LIN {X 0,Y 523.97,Z 254.844,A -85,B 0,C 180,E1 -4887.998,E2 -4887.998} C_VEL
LIN {X 0,Y 523.943,Z 254.846,A -85,B 0,C 180,E1 -4890.854,E2 -4890.854} C_VEL
LIN {X 0,Y 523.959,Z 254.847,A -85,B 0,C 180,E1 -4893.734,E2 -4893.734} C_VEL
LIN {X 0,Y 523.92,Z 254.85,A -85,B 0,C 180,E1 -4896.403,E2 -4896.403} C_VEL
LIN {X 0,Y 523.92,Z 254.85,A -85,B 0,C 180,E1 -4899.083,E2 -4899.083} C_VEL
LIN {X 0,Y 523.953,Z 254.847,A -85,B 0,C 180,E1 -4902.117,E2 -4902.117} C_VEL
LIN {X 0,Y 523.951,Z 254.848,A -85,B 0,C 180,E1 -4905.307,E2 -4905.307} C_VEL
LIN {X 0,Y 523.918,Z 254.849,A -85,B 0,C 180,E1 -4906.91,E2 -4906.91} C_VEL
LIN {X 0,Y 523.255,Z 254.934,A -85,B 0,C 180,E1 -4907.551,E2 -4907.551} C_VEL
LIN {X 0,Y 520.425,Z 255.289,A -85,B 0,C 180,E1 -4908.593,E2 -4908.593} C_VEL
LIN {X 0,Y 518.027,Z 255.589,A -85,B 0,C 180,E1 -4909.432,E2 -4909.432} C_VEL
LIN {X 0,Y 516.986,Z 255.716,A -85,B 0,C 180,E1 -4910.08,E2 -4910.08} C_VEL
LIN {X 0,Y 516.896,Z 255.726,A -85,B 0,C 180,E1 -4910.299,E2 -4910.299} C_VEL
LIN {X 0,Y 516.879,Z 255.727,A -85,B 0,C 180,E1 -4913.34,E2 -4913.34} C_VEL
LIN {X 0,Y 516.905,Z 255.724,A -85,B 0,C 180,E1 -4916.12,E2 -4916.12} C_VEL
LIN {X 0,Y 516.887,Z 255.727,A -85,B 0,C 180,E1 -4918.934,E2 -4918.934} C_VEL
LIN {X 0,Y 516.917,Z 255.723,A -85,B 0,C 180,E1 -4921.584,E2 -4921.584} C_VEL
LIN {X 0,Y 516.925,Z 255.721,A -85,B 0,C 180,E1 -4924.21,E2 -4924.21} C_VEL
LIN {X 0,Y 516.863,Z 255.727,A -85,B 0,C 180,E1 -4926.776,E2 -4926.776} C_VEL
LIN {X 0,Y 516.93,Z 255.721,A -85,B 0,C 180,E1 -4929.73,E2 -4929.73} C_VEL
LIN {X 0,Y 516.922,Z 255.722,A -85,B 0,C 180,E1 -4932.595,E2 -4932.595} C_VEL
LIN {X 0,Y 516.94,Z 255.719,A -85,B 0,C 180,E1 -4935.03,E2 -4935.03} C_VEL
LIN {X 0,Y 516.994,Z 255.712,A -85,B 0,C 180,E1 -4938.234,E2 -4938.234} C_VEL
LIN {X 0,Y 516.964,Z 255.717,A -85,B 0,C 180,E1 -4941.399,E2 -4941.399} C_VEL
LIN {X 0,Y 517.001,Z 255.713,A -85,B 0,C 180,E1 -4943.756,E2 -4943.756} C_VEL
LIN {X 0,Y 516.718,Z 255.749,A -85,B 0,C 180,E1 -4946.1,E2 -4946.1} C_VEL
LIN {X 0,Y 516.592,Z 255.877,A -85,B 0,C 180,E1 -4947.66,E2 -4947.66} C_VEL
LIN {X 0,Y 516.81,Z 258.103,A -85,B 0,C 180,E1 -4949.999,E2 -4949.999} C_VEL
LIN {X 0,Y 516.55,Z 261.858,A -85,B 0,C 180,E1 -4953.9,E2 -4953.9} C_VEL
LIN {X 0,Y 516.473,Z 264.87,A -85,B 0,C 180,E1 -4957.034,E2 -4957.034} C_VEL
LIN {X 0,Y 516.409,Z 267.914,A -85,B 0,C 180,E1 -4960.19,E2 -4960.19} C_VEL
LIN {X 0,Y 516.387,Z 270.207,A -85,B 0,C 180,E1 -4962.577,E2 -4962.577} C_VEL
LIN {X 0,Y 516.346,Z 271.07,A -85,B 0,C 180,E1 -4963.453,E2 -4963.453} C_VEL
LIN {X 0,Y 520.193,Z 284.754,A -85,B 0,C 180,E1 -4963.9,E2 -4963.9} C_VEL
LIN {X 0,Y 520.737,Z 287.139,A -85,B 0,C 180,E1 -4963.984,E2 -4963.984} C_VEL
LIN {X 0,Y 520.379,Z 301.279,A -85,B 0,C 180,E1 -4964.418,E2 -4964.418} C_VEL
LIN {X 0,Y 519.918,Z 315.967,A -85,B 0,C 180,E1 -4965.032,E2 -4965.032} C_VEL
LIN {X 0,Y 519.498,Z 328.44,A -85,B 0,C 180,E1 -4965.697,E2 -4965.697} C_VEL
LIN {X 0,Y 519.047,Z 341.031,A -85,B 0,C 180,E1 -4966.519,E2 -4966.519} C_VEL
LIN {X 0,Y 518.554,Z 352.891,A -85,B 0,C 180,E1 -4967.449,E2 -4967.449} C_VEL
LIN {X 0,Y 518.04,Z 364.714,A -85,B 0,C 180,E1 -4968.557,E2 -4968.557} C_VEL
LIN {X 0,Y 517.549,Z 376.157,A -85,B 0,C 180,E1 -4969.845,E2 -4969.845} C_VEL
LIN {X 0,Y 517.19,Z 385.528,A -85,B 0,C 180,E1 -4971.106,E2 -4971.106} C_VEL
LIN {X 0,Y 516.848,Z 394.593,A -85,B 0,C 180,E1 -4972.568,E2 -4972.568} C_VEL
LIN {X 0,Y 516.611,Z 402.308,A -85,B 0,C 180,E1 -4974.086,E2 -4974.086} C_VEL
LIN {X 0,Y 516.475,Z 407.75,A -85,B 0,C 180,E1 -4975.381,E2 -4975.381} C_VEL
LIN {X 0,Y 516.327,Z 413.495,A -85,B 0,C 180,E1 -4977.128,E2 -4977.128} C_VEL
LIN {X 0,Y 516.24,Z 416.777,A -85,B 0,C 180,E1 -4978.455,E2 -4978.455} C_VEL
LIN {X 0,Y 516.227,Z 418.584,A -85,B 0,C 180,E1 -4979.392,E2 -4979.392} C_VEL
LIN {X 0,Y 516.165,Z 420.848,A -85,B 0,C 180,E1 -4981.157,E2 -4981.157} C_VEL
LIN {X 0,Y 516.166,Z 421.563,A -85,B 0,C 180,E1 -4982.419,E2 -4982.419} C_VEL
LIN {X 0,Y 516.163,Z 421.505,A -85,B 0,C 180,E1 -4983.934,E2 -4983.934} C_VEL
LIN {X 0,Y 516.161,Z 420.566,A -85,B 0,C 180,E1 -4985.221,E2 -4985.221} C_VEL
LIN {X 0,Y 516.178,Z 418.411,A -85,B 0,C 180,E1 -4986.803,E2 -4986.803} C_VEL
LIN {X 0,Y 516.31,Z 415.336,A -85,B 0,C 180,E1 -4988.277,E2 -4988.277} C_VEL
LIN {X 0,Y 516.374,Z 411.065,A -85,B 0,C 180,E1 -4989.767,E2 -4989.767} C_VEL
LIN {X 0,Y 516.469,Z 405.957,A -85,B 0,C 180,E1 -4991.167,E2 -4991.167} C_VEL
LIN {X 0,Y 516.694,Z 398.838,A -85,B 0,C 180,E1 -4992.737,E2 -4992.737} C_VEL
LIN {X 0,Y 517.005,Z 390.921,A -85,B 0,C 180,E1 -4994.159,E2 -4994.159} C_VEL
LIN {X 0,Y 517.345,Z 381.995,A -85,B 0,C 180,E1 -4995.497,E2 -4995.497} C_VEL
LIN {X 0,Y 517.719,Z 372.189,A -85,B 0,C 180,E1 -4996.735,E2 -4996.735} C_VEL
LIN {X 0,Y 518.239,Z 360.952,A -85,B 0,C 180,E1 -4997.922,E2 -4997.922} C_VEL
LIN {X 0,Y 518.715,Z 350.053,A -85,B 0,C 180,E1 -4998.895,E2 -4998.895} C_VEL
LIN {X 0,Y 519.286,Z 336.91,A -85,B 0,C 180,E1 -4999.87,E2 -4999.87} C_VEL
LIN {X 0,Y 519.784,Z 322.543,A -85,B 0,C 180,E1 -5000.734,E2 -5000.734} C_VEL
LIN {X 0,Y 520.24,Z 308.093,A -85,B 0,C 180,E1 -5001.415,E2 -5001.415} C_VEL
LIN {X 0,Y 520.598,Z 293.591,A -85,B 0,C 180,E1 -5001.933,E2 -5001.933} C_VEL
LIN {X 0,Y 520.56,Z 286.17,A -85,B 0,C 180,E1 -5002.145,E2 -5002.145} C_VEL
LIN {X 0,Y 517.771,Z 276.119,A -85,B 0,C 180,E1 -5002.476,E2 -5002.476} C_VEL
LIN {X 0,Y 516.369,Z 271.47,A -85,B 0,C 180,E1 -5002.633,E2 -5002.633} C_VEL
LIN {X 0,Y 516.417,Z 269.147,A -85,B 0,C 180,E1 -5005.141,E2 -5005.141} C_VEL
LIN {X 0,Y 516.47,Z 266.567,A -85,B 0,C 180,E1 -5007.948,E2 -5007.948} C_VEL
LIN {X 0,Y 516.557,Z 264.068,A -85,B 0,C 180,E1 -5010.674,E2 -5010.674} C_VEL
LIN {X 0,Y 516.56,Z 261.657,A -85,B 0,C 180,E1 -5013.323,E2 -5013.323} C_VEL
LIN {X 0,Y 516.681,Z 259.257,A -85,B 0,C 180,E1 -5015.918,E2 -5015.918} C_VEL
LIN {X 0,Y 516.642,Z 256.888,A -85,B 0,C 180,E1 -5018.453,E2 -5018.453} C_VEL
LIN {X 0,Y 516.705,Z 255.752,A -85,B 0,C 180,E1 -5019.8,E2 -5019.8} C_VEL
LIN {X 0,Y 516.891,Z 255.729,A -85,B 0,C 180,E1 -5022.596,E2 -5022.596} C_VEL
LIN {X 0,Y 516.935,Z 255.721,A -85,B 0,C 180,E1 -5025.031,E2 -5025.031} C_VEL
LIN {X 0,Y 516.959,Z 255.717,A -85,B 0,C 180,E1 -5028.235,E2 -5028.235} C_VEL
LIN {X 0,Y 516.965,Z 255.716,A -85,B 0,C 180,E1 -5031.401,E2 -5031.401} C_VEL
LIN {X 0,Y 517.006,Z 255.712,A -85,B 0,C 180,E1 -5033.758,E2 -5033.758} C_VEL
LIN {X 0,Y 517.081,Z 255.701,A -85,B 0,C 180,E1 -5037.664,E2 -5037.664} C_VEL
LIN {X 0,Y 517.09,Z 255.701,A -85,B 0,C 180,E1 -5040.78,E2 -5040.78} C_VEL
LIN {X 0,Y 517.011,Z 255.711,A -85,B 0,C 180,E1 -5043.118,E2 -5043.118} C_VEL
LIN {X 0,Y 517.007,Z 255.71,A -85,B 0,C 180,E1 -5046.244,E2 -5046.244} C_VEL
LIN {X 0,Y 516.953,Z 255.718,A -85,B 0,C 180,E1 -5049.39,E2 -5049.39} C_VEL
LIN {X 0,Y 516.949,Z 255.719,A -85,B 0,C 180,E1 -5051.808,E2 -5051.808} C_VEL
LIN {X 0,Y 516.941,Z 255.719,A -85,B 0,C 180,E1 -5055.147,E2 -5055.147} C_VEL
LIN {X 0,Y 516.922,Z 255.723,A -85,B 0,C 180,E1 -5058.223,E2 -5058.223} C_VEL
LIN {X 0,Y 516.911,Z 255.723,A -85,B 0,C 180,E1 -5060.702,E2 -5060.702} C_VEL
LIN {X 0,Y 516.909,Z 255.723,A -85,B 0,C 180,E1 -5064.073,E2 -5064.073} C_VEL
LIN {X 0,Y 516.927,Z 255.723,A -85,B 0,C 180,E1 -5066.658,E2 -5066.658} C_VEL
LIN {X 0,Y 516.909,Z 255.725,A -85,B 0,C 180,E1 -5069.524,E2 -5069.524} C_VEL
LIN {X 0,Y 516.893,Z 255.728,A -85,B 0,C 180,E1 -5072.544,E2 -5072.544} C_VEL
LIN {X 0,Y 516.864,Z 255.733,A -85,B 0,C 180,E1 -5075.33,E2 -5075.33} C_VEL
LIN {X 0,Y 516.879,Z 255.73,A -85,B 0,C 180,E1 -5077.944,E2 -5077.944} C_VEL
LIN {X 0,Y 516.883,Z 255.729,A -85,B 0,C 180,E1 -5080.742,E2 -5080.742} C_VEL
LIN {X 0,Y 516.882,Z 255.729,A -85,B 0,C 180,E1 -5082.832,E2 -5082.832} C_VEL
LIN {X 0,Y 516.93,Z 255.773,A -85,B 0,C 180,E1 -5084.578,E2 -5084.578} C_VEL
LIN {X 0,Y 517.92,Z 261.24,A -85,B 0,C 180,E1 -5087.119,E2 -5087.119} C_VEL
LIN {X 0,Y 518.273,Z 265.231,A -85,B 0,C 180,E1 -5088.878,E2 -5088.878} C_VEL
LIN {X 0,Y 518.125,Z 271.563,A -85,B 0,C 180,E1 -5091.395,E2 -5091.395} C_VEL
LIN {X 0,Y 517.889,Z 277.824,A -85,B 0,C 180,E1 -5093.821,E2 -5093.821} C_VEL
LIN {X 0,Y 517.701,Z 286.966,A -85,B 0,C 180,E1 -5097.112,E2 -5097.112} C_VEL
LIN {X 0,Y 517.53,Z 294.866,A -85,B 0,C 180,E1 -5099.838,E2 -5099.838} C_VEL
LIN {X 0,Y 517.327,Z 302.394,A -85,B 0,C 180,E1 -5102.491,E2 -5102.491} C_VEL
LIN {X 0,Y 517.143,Z 309.82,A -85,B 0,C 180,E1 -5105.085,E2 -5105.085} C_VEL
LIN {X 0,Y 516.963,Z 318.485,A -85,B 0,C 180,E1 -5108.047,E2 -5108.047} C_VEL
LIN {X 0,Y 516.826,Z 325.427,A -85,B 0,C 180,E1 -5110.378,E2 -5110.378} C_VEL
LIN {X 0,Y 520.774,Z 341.818,A -85,B 0,C 180,E1 -5110.836,E2 -5110.836} C_VEL
LIN {X 0,Y 520.392,Z 356.97,A -85,B 0,C 180,E1 -5111.264,E2 -5111.264} C_VEL
LIN {X 0,Y 520.029,Z 371.072,A -85,B 0,C 180,E1 -5111.817,E2 -5111.817} C_VEL
LIN {X 0,Y 519.548,Z 384.377,A -85,B 0,C 180,E1 -5112.484,E2 -5112.484} C_VEL
LIN {X 0,Y 519.048,Z 397.209,A -85,B 0,C 180,E1 -5113.279,E2 -5113.279} C_VEL
LIN {X 0,Y 518.531,Z 410.363,A -85,B 0,C 180,E1 -5114.272,E2 -5114.272} C_VEL
LIN {X 0,Y 518.039,Z 421.386,A -85,B 0,C 180,E1 -5115.264,E2 -5115.264} C_VEL
LIN {X 0,Y 517.634,Z 432.514,A -85,B 0,C 180,E1 -5116.456,E2 -5116.456} C_VEL
LIN {X 0,Y 517.156,Z 443.311,A -85,B 0,C 180,E1 -5117.841,E2 -5117.841} C_VEL
LIN {X 0,Y 516.912,Z 452.298,A -85,B 0,C 180,E1 -5119.226,E2 -5119.226} C_VEL
LIN {X 0,Y 516.637,Z 459.753,A -85,B 0,C 180,E1 -5120.606,E2 -5120.606} C_VEL
LIN {X 0,Y 516.463,Z 466.703,A -85,B 0,C 180,E1 -5122.18,E2 -5122.18} C_VEL
LIN {X 0,Y 516.36,Z 472.164,A -85,B 0,C 180,E1 -5123.75,E2 -5123.75} C_VEL
LIN {X 0,Y 516.239,Z 476.293,A -85,B 0,C 180,E1 -5125.315,E2 -5125.315} C_VEL
LIN {X 0,Y 516.272,Z 479.187,A -85,B 0,C 180,E1 -5126.879,E2 -5126.879} C_VEL
LIN {X 0,Y 516.189,Z 480.911,A -85,B 0,C 180,E1 -5128.44,E2 -5128.44} C_VEL
LIN {X 0,Y 516.151,Z 481.5,A -85,B 0,C 180,E1 -5130.001,E2 -5130.001} C_VEL
LIN {X 0,Y 516.189,Z 480.909,A -85,B 0,C 180,E1 -5131.561,E2 -5131.561} C_VEL
LIN {X 0,Y 516.272,Z 479.182,A -85,B 0,C 180,E1 -5133.122,E2 -5133.122} C_VEL
LIN {X 0,Y 516.239,Z 476.289,A -85,B 0,C 180,E1 -5134.686,E2 -5134.686} C_VEL
LIN {X 0,Y 516.352,Z 472.163,A -85,B 0,C 180,E1 -5136.252,E2 -5136.252} C_VEL
LIN {X 0,Y 516.464,Z 466.699,A -85,B 0,C 180,E1 -5137.822,E2 -5137.822} C_VEL
LIN {X 0,Y 516.638,Z 459.744,A -85,B 0,C 180,E1 -5139.396,E2 -5139.396} C_VEL
LIN {X 0,Y 516.973,Z 451.082,A -85,B 0,C 180,E1 -5140.972,E2 -5140.972} C_VEL
LIN {X 0,Y 517.228,Z 442.019,A -85,B 0,C 180,E1 -5142.338,E2 -5142.338} C_VEL
LIN {X 0,Y 517.635,Z 432.504,A -85,B 0,C 180,E1 -5143.545,E2 -5143.545} C_VEL
LIN {X 0,Y 518.095,Z 420.35,A -85,B 0,C 180,E1 -5144.836,E2 -5144.836} C_VEL
LIN {X 0,Y 518.628,Z 408.21,A -85,B 0,C 180,E1 -5145.907,E2 -5145.907} C_VEL
LIN {X 0,Y 519.087,Z 395.767,A -85,B 0,C 180,E1 -5146.822,E2 -5146.822} C_VEL
LIN {X 0,Y 519.577,Z 382.586,A -85,B 0,C 180,E1 -5147.618,E2 -5147.618} C_VEL
LIN {X 0,Y 520.083,Z 369.43,A -85,B 0,C 180,E1 -5148.255,E2 -5148.255} C_VEL
LIN {X 0,Y 520.483,Z 354.499,A -85,B 0,C 180,E1 -5148.816,E2 -5148.816} C_VEL
LIN {X 0,Y 520.673,Z 341.239,A -85,B 0,C 180,E1 -5149.182,E2 -5149.182} C_VEL
LIN {X 0,Y 516.823,Z 325.426,A -85,B 0,C 180,E1 -5149.622,E2 -5149.622} C_VEL
LIN {X 0,Y 516.971,Z 317.119,A -85,B 0,C 180,E1 -5152.417,E2 -5152.417} C_VEL
LIN {X 0,Y 517.188,Z 308.579,A -85,B 0,C 180,E1 -5155.344,E2 -5155.344} C_VEL
LIN {X 0,Y 517.427,Z 299.915,A -85,B 0,C 180,E1 -5158.385,E2 -5158.385} C_VEL
LIN {X 0,Y 517.554,Z 291.891,A -85,B 0,C 180,E1 -5161.185,E2 -5161.185} C_VEL
LIN {X 0,Y 517.817,Z 283.8,A -85,B 0,C 180,E1 -5164.115,E2 -5164.115} C_VEL
LIN {X 0,Y 518.095,Z 275.662,A -85,B 0,C 180,E1 -5167.183,E2 -5167.183} C_VEL
LIN {X 0,Y 518.293,Z 268.202,A -85,B 0,C 180,E1 -5170.092,E2 -5170.092} C_VEL
LIN {X 0,Y 518.181,Z 263.095,A -85,B 0,C 180,E1 -5172.194,E2 -5172.194} C_VEL
LIN {X 0,Y 517.331,Z 257.986,A -85,B 0,C 180,E1 -5174.503,E2 -5174.503} C_VEL
LIN {X 0,Y 516.923,Z 255.721,A -85,B 0,C 180,E1 -5175.626,E2 -5175.626} C_VEL
LIN {X 0,Y 516.918,Z 255.724,A -85,B 0,C 180,E1 -5178.399,E2 -5178.399} C_VEL
LIN {X 0,Y 516.885,Z 255.727,A -85,B 0,C 180,E1 -5181.284,E2 -5181.284} C_VEL
LIN {X 0,Y 516.876,Z 255.727,A -85,B 0,C 180,E1 -5184.22,E2 -5184.22} C_VEL
LIN {X 0,Y 516.886,Z 255.727,A -85,B 0,C 180,E1 -5187.052,E2 -5187.052} C_VEL
LIN {X 0,Y 516.897,Z 255.725,A -85,B 0,C 180,E1 -5189.796,E2 -5189.796} C_VEL
LIN {X 0,Y 516.932,Z 255.721,A -85,B 0,C 180,E1 -5192.467,E2 -5192.467} C_VEL
LIN {X 0,Y 516.914,Z 255.724,A -85,B 0,C 180,E1 -5195.072,E2 -5195.072} C_VEL
LIN {X 0,Y 516.892,Z 255.727,A -85,B 0,C 180,E1 -5198.462,E2 -5198.462} C_VEL
LIN {X 0,Y 516.909,Z 255.724,A -85,B 0,C 180,E1 -5200.954,E2 -5200.954} C_VEL
LIN {X 0,Y 516.919,Z 255.722,A -85,B 0,C 180,E1 -5203.41,E2 -5203.41} C_VEL
LIN {X 0,Y 516.899,Z 255.725,A -85,B 0,C 180,E1 -5205.833,E2 -5205.833} C_VEL
LIN {X 0,Y 516.971,Z 255.716,A -85,B 0,C 180,E1 -5208.233,E2 -5208.233} C_VEL
LIN {X 0,Y 516.971,Z 255.715,A -85,B 0,C 180,E1 -5211.399,E2 -5211.399} C_VEL
LIN {X 0,Y 517.028,Z 255.709,A -85,B 0,C 180,E1 -5214.539,E2 -5214.539} C_VEL
LIN {X 0,Y 517.088,Z 255.7,A -85,B 0,C 180,E1 -5217.662,E2 -5217.662} C_VEL
LIN {X 0,Y 517.098,Z 255.7,A -85,B 0,C 180,E1 -5220.778,E2 -5220.778} C_VEL
LIN {X 0,Y 517.015,Z 255.711,A -85,B 0,C 180,E1 -5223.116,E2 -5223.116} C_VEL
LIN {X 0,Y 517.012,Z 255.711,A -85,B 0,C 180,E1 -5226.242,E2 -5226.242} C_VEL
LIN {X 0,Y 516.954,Z 255.717,A -85,B 0,C 180,E1 -5229.388,E2 -5229.388} C_VEL
LIN {X 0,Y 516.955,Z 255.719,A -85,B 0,C 180,E1 -5231.806,E2 -5231.806} C_VEL
LIN {X 0,Y 516.947,Z 255.717,A -85,B 0,C 180,E1 -5235.145,E2 -5235.145} C_VEL
LIN {X 0,Y 516.927,Z 255.722,A -85,B 0,C 180,E1 -5238.221,E2 -5238.221} C_VEL
LIN {X 0,Y 516.913,Z 255.723,A -85,B 0,C 180,E1 -5240.7,E2 -5240.7} C_VEL
LIN {X 0,Y 516.912,Z 255.724,A -85,B 0,C 180,E1 -5244.071,E2 -5244.071} C_VEL
LIN {X 0,Y 516.926,Z 255.721,A -85,B 0,C 180,E1 -5246.656,E2 -5246.656} C_VEL
LIN {X 0,Y 516.91,Z 255.724,A -85,B 0,C 180,E1 -5249.523,E2 -5249.523} C_VEL
LIN {X 0,Y 516.896,Z 255.726,A -85,B 0,C 180,E1 -5252.543,E2 -5252.543} C_VEL
LIN {X 0,Y 516.881,Z 255.726,A -85,B 0,C 180,E1 -5255.331,E2 -5255.331} C_VEL
LIN {X 0,Y 516.879,Z 255.729,A -85,B 0,C 180,E1 -5257.942,E2 -5257.942} C_VEL
LIN {X 0,Y 516.882,Z 255.727,A -85,B 0,C 180,E1 -5260.74,E2 -5260.74} C_VEL
LIN {X 0,Y 516.9,Z 255.724,A -85,B 0,C 180,E1 -5262.828,E2 -5262.828} C_VEL
LIN {X 0,Y 516.918,Z 255.722,A -85,B 0,C 180,E1 -5265.009,E2 -5265.009} C_VEL
LIN {X 0,Y 516.917,Z 255.722,A -85,B 0,C 180,E1 -5268.396,E2 -5268.396} C_VEL
LIN {X 0,Y 516.896,Z 255.726,A -85,B 0,C 180,E1 -5270.299,E2 -5270.299} C_VEL
LIN {X 0,Y 516.215,Z 255.809,A -85,B 0,C 180,E1 -5270.949,E2 -5270.949} C_VEL
LIN {X 0,Y 513.362,Z 256.166,A -85,B 0,C 180,E1 -5272.004,E2 -5272.004} C_VEL
LIN {X 0,Y 510.954,Z 256.469,A -85,B 0,C 180,E1 -5272.855,E2 -5272.855} C_VEL
LIN {X 0,Y 509.914,Z 256.597,A -85,B 0,C 180,E1 -5273.511,E2 -5273.511} C_VEL
LIN {X 0,Y 509.826,Z 256.607,A -85,B 0,C 180,E1 -5273.733,E2 -5273.733} C_VEL
LIN {X 0,Y 509.855,Z 256.602,A -85,B 0,C 180,E1 -5276.538,E2 -5276.538} C_VEL
LIN {X 0,Y 509.843,Z 256.604,A -85,B 0,C 180,E1 -5279.334,E2 -5279.334} C_VEL
LIN {X 0,Y 509.888,Z 256.598,A -85,B 0,C 180,E1 -5282.054,E2 -5282.054} C_VEL
LIN {X 0,Y 509.87,Z 256.599,A -85,B 0,C 180,E1 -5284.703,E2 -5284.703} C_VEL
LIN {X 0,Y 509.847,Z 256.604,A -85,B 0,C 180,E1 -5287.449,E2 -5287.449} C_VEL
LIN {X 0,Y 509.908,Z 256.596,A -85,B 0,C 180,E1 -5289.844,E2 -5289.844} C_VEL
LIN {X 0,Y 509.878,Z 256.6,A -85,B 0,C 180,E1 -5293.174,E2 -5293.174} C_VEL
LIN {X 0,Y 509.864,Z 256.602,A -85,B 0,C 180,E1 -5295.634,E2 -5295.634} C_VEL
LIN {X 0,Y 509.916,Z 256.595,A -85,B 0,C 180,E1 -5298.874,E2 -5298.874} C_VEL
LIN {X 0,Y 509.942,Z 256.59,A -85,B 0,C 180,E1 -5302.078,E2 -5302.078} C_VEL
LIN {X 0,Y 509.943,Z 256.589,A -85,B 0,C 180,E1 -5304.463,E2 -5304.463} C_VEL
LIN {X 0,Y 509.534,Z 256.645,A -85,B 0,C 180,E1 -5307.628,E2 -5307.628} C_VEL
LIN {X 0,Y 509.795,Z 258.058,A -85,B 0,C 180,E1 -5309.21,E2 -5309.21} C_VEL
LIN {X 0,Y 509.474,Z 260.352,A -85,B 0,C 180,E1 -5311.58,E2 -5311.58} C_VEL
LIN {X 0,Y 509.465,Z 263.372,A -85,B 0,C 180,E1 -5314.747,E2 -5314.747} C_VEL
LIN {X 0,Y 509.418,Z 265.644,A -85,B 0,C 180,E1 -5317.132,E2 -5317.132} C_VEL
LIN {X 0,Y 509.344,Z 268.73,A -85,B 0,C 180,E1 -5320.333,E2 -5320.333} C_VEL
LIN {X 0,Y 509.292,Z 271.48,A -85,B 0,C 180,E1 -5323.186,E2 -5323.186} C_VEL
LIN {X 0,Y 513.52,Z 286.197,A -85,B 0,C 180,E1 -5323.67,E2 -5323.67} C_VEL
LIN {X 0,Y 513.979,Z 288.927,A -85,B 0,C 180,E1 -5323.766,E2 -5323.766} C_VEL
LIN {X 0,Y 513.576,Z 304.035,A -85,B 0,C 180,E1 -5324.259,E2 -5324.259} C_VEL
LIN {X 0,Y 513.1,Z 318.162,A -85,B 0,C 180,E1 -5324.881,E2 -5324.881} C_VEL
LIN {X 0,Y 512.637,Z 331.194,A -85,B 0,C 180,E1 -5325.607,E2 -5325.607} C_VEL
LIN {X 0,Y 512.081,Z 345.219,A -85,B 0,C 180,E1 -5326.578,E2 -5326.578} C_VEL
LIN {X 0,Y 511.549,Z 357.293,A -85,B 0,C 180,E1 -5327.592,E2 -5327.592} C_VEL
LIN {X 0,Y 511.012,Z 367.896,A -85,B 0,C 180,E1 -5328.648,E2 -5328.648} C_VEL
LIN {X 0,Y 510.55,Z 378.603,A -85,B 0,C 180,E1 -5329.919,E2 -5329.919} C_VEL
LIN {X 0,Y 510.119,Z 387.673,A -85,B 0,C 180,E1 -5331.201,E2 -5331.201} C_VEL
LIN {X 0,Y 509.798,Z 396.556,A -85,B 0,C 180,E1 -5332.705,E2 -5332.705} C_VEL
LIN {X 0,Y 509.575,Z 402.926,A -85,B 0,C 180,E1 -5334.007,E2 -5334.007} C_VEL
LIN {X 0,Y 509.418,Z 408.335,A -85,B 0,C 180,E1 -5335.32,E2 -5335.32} C_VEL
LIN {X 0,Y 509.287,Z 412.746,A -85,B 0,C 180,E1 -5336.646,E2 -5336.646} C_VEL
LIN {X 0,Y 509.195,Z 416.312,A -85,B 0,C 180,E1 -5337.986,E2 -5337.986} C_VEL
LIN {X 0,Y 509.131,Z 419.721,A -85,B 0,C 180,E1 -5339.797,E2 -5339.797} C_VEL
LIN {X 0,Y 509.089,Z 421.296,A -85,B 0,C 180,E1 -5341.142,E2 -5341.142} C_VEL
LIN {X 0,Y 509.072,Z 422.049,A -85,B 0,C 180,E1 -5342.636,E2 -5342.636} C_VEL
LIN {X 0,Y 509.095,Z 421.64,A -85,B 0,C 180,E1 -5344.471,E2 -5344.471} C_VEL
LIN {X 0,Y 509.073,Z 420.803,A -85,B 0,C 180,E1 -5345.462,E2 -5345.462} C_VEL
LIN {X 0,Y 509.109,Z 418.94,A -85,B 0,C 180,E1 -5346.809,E2 -5346.809} C_VEL
LIN {X 0,Y 509.251,Z 415.678,A -85,B 0,C 180,E1 -5348.39,E2 -5348.39} C_VEL
LIN {X 0,Y 509.34,Z 411.357,A -85,B 0,C 180,E1 -5349.912,E2 -5349.912} C_VEL
LIN {X 0,Y 509.461,Z 405.675,A -85,B 0,C 180,E1 -5351.464,E2 -5351.464} C_VEL
LIN {X 0,Y 509.715,Z 398.396,A -85,B 0,C 180,E1 -5353.051,E2 -5353.051} C_VEL
LIN {X 0,Y 510.048,Z 390.848,A -85,B 0,C 180,E1 -5354.399,E2 -5354.399} C_VEL
LIN {X 0,Y 510.428,Z 382.045,A -85,B 0,C 180,E1 -5355.723,E2 -5355.723} C_VEL
LIN {X 0,Y 510.86,Z 371.824,A -85,B 0,C 180,E1 -5357.014,E2 -5357.014} C_VEL
LIN {X 0,Y 511.407,Z 360.57,A -85,B 0,C 180,E1 -5358.204,E2 -5358.204} C_VEL
LIN {X 0,Y 511.945,Z 349.159,A -85,B 0,C 180,E1 -5359.218,E2 -5359.218} C_VEL
LIN {X 0,Y 512.5,Z 336.309,A -85,B 0,C 180,E1 -5360.168,E2 -5360.168} C_VEL
LIN {X 0,Y 513.037,Z 323.002,A -85,B 0,C 180,E1 -5360.971,E2 -5360.971} C_VEL
LIN {X 0,Y 513.52,Z 308.765,A -85,B 0,C 180,E1 -5361.652,E2 -5361.652} C_VEL
LIN {X 0,Y 513.923,Z 293.692,A -85,B 0,C 180,E1 -5362.196,E2 -5362.196} C_VEL
LIN {X 0,Y 513.81,Z 287.32,A -85,B 0,C 180,E1 -5362.384,E2 -5362.384} C_VEL
LIN {X 0,Y 510.983,Z 277.314,A -85,B 0,C 180,E1 -5362.73,E2 -5362.73} C_VEL
LIN {X 0,Y 509.309,Z 271.968,A -85,B 0,C 180,E1 -5362.903,E2 -5362.903} C_VEL
LIN {X 0,Y 509.363,Z 269.219,A -85,B 0,C 180,E1 -5365.878,E2 -5365.878} C_VEL
LIN {X 0,Y 509.457,Z 266.557,A -85,B 0,C 180,E1 -5368.791,E2 -5368.791} C_VEL
LIN {X 0,Y 509.499,Z 263.615,A -85,B 0,C 180,E1 -5372.032,E2 -5372.032} C_VEL
LIN {X 0,Y 509.542,Z 261.186,A -85,B 0,C 180,E1 -5374.687,E2 -5374.687} C_VEL
LIN {X 0,Y 509.59,Z 258.574,A -85,B 0,C 180,E1 -5377.521,E2 -5377.521} C_VEL
LIN {X 0,Y 509.677,Z 256.627,A -85,B 0,C 180,E1 -5379.836,E2 -5379.836} C_VEL
LIN {X 0,Y 509.855,Z 256.606,A -85,B 0,C 180,E1 -5382.348,E2 -5382.348} C_VEL
LIN {X 0,Y 509.903,Z 256.597,A -85,B 0,C 180,E1 -5384.82,E2 -5384.82} C_VEL
LIN {X 0,Y 509.895,Z 256.597,A -85,B 0,C 180,E1 -5388.124,E2 -5388.124} C_VEL
LIN {X 0,Y 509.912,Z 256.595,A -85,B 0,C 180,E1 -5391.281,E2 -5391.281} C_VEL
LIN {X 0,Y 509.974,Z 256.588,A -85,B 0,C 180,E1 -5393.671,E2 -5393.671} C_VEL
LIN {X 0,Y 510.052,Z 256.577,A -85,B 0,C 180,E1 -5397.632,E2 -5397.632} C_VEL
LIN {X 0,Y 510.06,Z 256.577,A -85,B 0,C 180,E1 -5400.79,E2 -5400.79} C_VEL
LIN {X 0,Y 509.953,Z 256.59,A -85,B 0,C 180,E1 -5403.161,E2 -5403.161} C_VEL
LIN {X 0,Y 509.975,Z 256.586,A -85,B 0,C 180,E1 -5406.33,E2 -5406.33} C_VEL
LIN {X 0,Y 509.914,Z 256.595,A -85,B 0,C 180,E1 -5408.721,E2 -5408.721} C_VEL
LIN {X 0,Y 509.901,Z 256.598,A -85,B 0,C 180,E1 -5411.932,E2 -5411.932} C_VEL
LIN {X 0,Y 509.891,Z 256.598,A -85,B 0,C 180,E1 -5415.243,E2 -5415.243} C_VEL
LIN {X 0,Y 509.885,Z 256.598,A -85,B 0,C 180,E1 -5418.002,E2 -5418.002} C_VEL
LIN {X 0,Y 509.849,Z 256.602,A -85,B 0,C 180,E1 -5421.002,E2 -5421.002} C_VEL
LIN {X 0,Y 509.835,Z 256.605,A -85,B 0,C 180,E1 -5423.564,E2 -5423.564} C_VEL
LIN {X 0,Y 509.912,Z 256.596,A -85,B 0,C 180,E1 -5426.38,E2 -5426.38} C_VEL
LIN {X 0,Y 509.875,Z 256.602,A -85,B 0,C 180,E1 -5428.845,E2 -5428.845} C_VEL
LIN {X 0,Y 509.817,Z 256.61,A -85,B 0,C 180,E1 -5431.591,E2 -5431.591} C_VEL
LIN {X 0,Y 509.845,Z 256.608,A -85,B 0,C 180,E1 -5434.414,E2 -5434.414} C_VEL
LIN {X 0,Y 509.815,Z 256.613,A -85,B 0,C 180,E1 -5437.341,E2 -5437.341} C_VEL
LIN {X 0,Y 509.836,Z 256.606,A -85,B 0,C 180,E1 -5440.383,E2 -5440.383} C_VEL
LIN {X 0,Y 509.822,Z 256.609,A -85,B 0,C 180,E1 -5443.063,E2 -5443.063} C_VEL
LIN {X 0,Y 509.859,Z 256.621,A -85,B 0,C 180,E1 -5444.212,E2 -5444.212} C_VEL
LIN {X 0,Y 510.86,Z 261.949,A -85,B 0,C 180,E1 -5446.814,E2 -5446.814} C_VEL
LIN {X 0,Y 511.314,Z 266.361,A -85,B 0,C 180,E1 -5448.719,E2 -5448.719} C_VEL
LIN {X 0,Y 511.148,Z 272.465,A -85,B 0,C 180,E1 -5451.23,E2 -5451.23} C_VEL
LIN {X 0,Y 510.909,Z 278.821,A -85,B 0,C 180,E1 -5453.737,E2 -5453.737} C_VEL
LIN {X 0,Y 510.676,Z 287.976,A -85,B 0,C 180,E1 -5457.087,E2 -5457.087} C_VEL
LIN {X 0,Y 510.47,Z 297.127,A -85,B 0,C 180,E1 -5460.289,E2 -5460.289} C_VEL
LIN {X 0,Y 510.293,Z 304.869,A -85,B 0,C 180,E1 -5462.968,E2 -5462.968} C_VEL
LIN {X 0,Y 510.057,Z 313.534,A -85,B 0,C 180,E1 -5466.017,E2 -5466.017} C_VEL
LIN {X 0,Y 509.883,Z 322.199,A -85,B 0,C 180,E1 -5469,E2 -5469} C_VEL
LIN {X 0,Y 509.781,Z 325.429,A -85,B 0,C 180,E1 -5470.096,E2 -5470.096} C_VEL
LIN {X 0,Y 513.785,Z 341.937,A -85,B 0,C 180,E1 -5470.567,E2 -5470.567} C_VEL
LIN {X 0,Y 513.991,Z 345.193,A -85,B 0,C 180,E1 -5470.657,E2 -5470.657} C_VEL
LIN {X 0,Y 513.657,Z 359.079,A -85,B 0,C 180,E1 -5471.081,E2 -5471.081} C_VEL
LIN {X 0,Y 513.169,Z 373.813,A -85,B 0,C 180,E1 -5471.692,E2 -5471.692} C_VEL
LIN {X 0,Y 512.613,Z 387.891,A -85,B 0,C 180,E1 -5472.446,E2 -5472.446} C_VEL
LIN {X 0,Y 512.032,Z 401.468,A -85,B 0,C 180,E1 -5473.351,E2 -5473.351} C_VEL
LIN {X 0,Y 511.536,Z 414.073,A -85,B 0,C 180,E1 -5474.376,E2 -5474.376} C_VEL
LIN {X 0,Y 510.962,Z 425.286,A -85,B 0,C 180,E1 -5475.463,E2 -5475.463} C_VEL
LIN {X 0,Y 510.504,Z 435.77,A -85,B 0,C 180,E1 -5476.669,E2 -5476.669} C_VEL
LIN {X 0,Y 510.002,Z 446.021,A -85,B 0,C 180,E1 -5478.071,E2 -5478.071} C_VEL
LIN {X 0,Y 509.818,Z 454.537,A -85,B 0,C 180,E1 -5479.476,E2 -5479.476} C_VEL
LIN {X 0,Y 509.536,Z 461.619,A -85,B 0,C 180,E1 -5480.874,E2 -5480.874} C_VEL
LIN {X 0,Y 509.352,Z 468.186,A -85,B 0,C 180,E1 -5482.469,E2 -5482.469} C_VEL
LIN {X 0,Y 509.297,Z 473.323,A -85,B 0,C 180,E1 -5484.06,E2 -5484.06} C_VEL
LIN {X 0,Y 509.159,Z 476.293,A -85,B 0,C 180,E1 -5485.25,E2 -5485.25} C_VEL
LIN {X 0,Y 509.188,Z 479.187,A -85,B 0,C 180,E1 -5486.836,E2 -5486.836} C_VEL
LIN {X 0,Y 509.11,Z 480.911,A -85,B 0,C 180,E1 -5488.418,E2 -5488.418} C_VEL
LIN {X 0,Y 509.063,Z 481.5,A -85,B 0,C 180,E1 -5490.001,E2 -5490.001} C_VEL
LIN {X 0,Y 509.11,Z 480.908,A -85,B 0,C 180,E1 -5491.583,E2 -5491.583} C_VEL
LIN {X 0,Y 509.189,Z 479.182,A -85,B 0,C 180,E1 -5493.165,E2 -5493.165} C_VEL
LIN {X 0,Y 509.159,Z 476.288,A -85,B 0,C 180,E1 -5494.751,E2 -5494.751} C_VEL
LIN {X 0,Y 509.262,Z 472.163,A -85,B 0,C 180,E1 -5496.339,E2 -5496.339} C_VEL
LIN {X 0,Y 509.386,Z 466.699,A -85,B 0,C 180,E1 -5497.931,E2 -5497.931} C_VEL
LIN {X 0,Y 509.561,Z 459.743,A -85,B 0,C 180,E1 -5499.527,E2 -5499.527} C_VEL
LIN {X 0,Y 509.956,Z 451.081,A -85,B 0,C 180,E1 -5501.125,E2 -5501.125} C_VEL
LIN {X 0,Y 510.24,Z 442.019,A -85,B 0,C 180,E1 -5502.51,E2 -5502.51} C_VEL
LIN {X 0,Y 510.654,Z 432.504,A -85,B 0,C 180,E1 -5503.734,E2 -5503.734} C_VEL
LIN {X 0,Y 511.181,Z 420.35,A -85,B 0,C 180,E1 -5505.041,E2 -5505.041} C_VEL
LIN {X 0,Y 511.747,Z 408.211,A -85,B 0,C 180,E1 -5506.127,E2 -5506.127} C_VEL
LIN {X 0,Y 512.274,Z 395.766,A -85,B 0,C 180,E1 -5507.053,E2 -5507.053} C_VEL
LIN {X 0,Y 512.789,Z 382.585,A -85,B 0,C 180,E1 -5507.859,E2 -5507.859} C_VEL
LIN {X 0,Y 513.399,Z 367.969,A -85,B 0,C 180,E1 -5508.568,E2 -5508.568} C_VEL
LIN {X 0,Y 513.798,Z 352.709,A -85,B 0,C 180,E1 -5509.131,E2 -5509.131} C_VEL
LIN {X 0,Y 513.944,Z 342.545,A -85,B 0,C 180,E1 -5509.413,E2 -5509.413} C_VEL
LIN {X 0,Y 509.999,Z 326.691,A -85,B 0,C 180,E1 -5509.876,E2 -5509.876} C_VEL
LIN {X 0,Y 509.8,Z 325.391,A -85,B 0,C 180,E1 -5509.916,E2 -5509.916} C_VEL
LIN {X 0,Y 509.929,Z 317.244,A -85,B 0,C 180,E1 -5512.7,E2 -5512.7} C_VEL
LIN {X 0,Y 510.188,Z 308.579,A -85,B 0,C 180,E1 -5515.717,E2 -5515.717} C_VEL
LIN {X 0,Y 510.46,Z 299.825,A -85,B 0,C 180,E1 -5518.809,E2 -5518.809} C_VEL
LIN {X 0,Y 510.634,Z 290.651,A -85,B 0,C 180,E1 -5521.998,E2 -5521.998} C_VEL
LIN {X 0,Y 510.854,Z 283.125,A -85,B 0,C 180,E1 -5524.815,E2 -5524.815} C_VEL
LIN {X 0,Y 511.174,Z 275.557,A -85,B 0,C 180,E1 -5527.722,E2 -5527.722} C_VEL
LIN {X 0,Y 511.322,Z 269.211,A -85,B 0,C 180,E1 -5530.241,E2 -5530.241} C_VEL
LIN {X 0,Y 511.208,Z 264.256,A -85,B 0,C 180,E1 -5532.349,E2 -5532.349} C_VEL
LIN {X 0,Y 510.351,Z 259.311,A -85,B 0,C 180,E1 -5534.614,E2 -5534.614} C_VEL
LIN {X 0,Y 509.86,Z 256.599,A -85,B 0,C 180,E1 -5535.941,E2 -5535.941} C_VEL
LIN {X 0,Y 509.86,Z 256.603,A -85,B 0,C 180,E1 -5538.574,E2 -5538.574} C_VEL
LIN {X 0,Y 509.856,Z 256.603,A -85,B 0,C 180,E1 -5541.786,E2 -5541.786} C_VEL
LIN {X 0,Y 509.835,Z 256.607,A -85,B 0,C 180,E1 -5544.622,E2 -5544.622} C_VEL
LIN {X 0,Y 509.865,Z 256.601,A -85,B 0,C 180,E1 -5547.481,E2 -5547.481} C_VEL
LIN {X 0,Y 509.864,Z 256.601,A -85,B 0,C 180,E1 -5550.274,E2 -5550.274} C_VEL
LIN {X 0,Y 509.89,Z 256.6,A -85,B 0,C 180,E1 -5552.944,E2 -5552.944} C_VEL
LIN {X 0,Y 509.87,Z 256.599,A -85,B 0,C 180,E1 -5555.573,E2 -5555.573} C_VEL
LIN {X 0,Y 509.856,Z 256.603,A -85,B 0,C 180,E1 -5558.998,E2 -5558.998} C_VEL
LIN {X 0,Y 509.895,Z 256.596,A -85,B 0,C 180,E1 -5561.999,E2 -5561.999} C_VEL
LIN {X 0,Y 509.916,Z 256.595,A -85,B 0,C 180,E1 -5564.818,E2 -5564.818} C_VEL
LIN {X 0,Y 509.906,Z 256.596,A -85,B 0,C 180,E1 -5568.124,E2 -5568.124} C_VEL
LIN {X 0,Y 509.917,Z 256.593,A -85,B 0,C 180,E1 -5571.279,E2 -5571.279} C_VEL
LIN {X 0,Y 509.978,Z 256.587,A -85,B 0,C 180,E1 -5574.463,E2 -5574.463} C_VEL
LIN {X 0,Y 510.059,Z 256.575,A -85,B 0,C 180,E1 -5577.63,E2 -5577.63} C_VEL
LIN {X 0,Y 510.069,Z 256.576,A -85,B 0,C 180,E1 -5580.789,E2 -5580.789} C_VEL
LIN {X 0,Y 509.957,Z 256.589,A -85,B 0,C 180,E1 -5583.159,E2 -5583.159} C_VEL
LIN {X 0,Y 509.981,Z 256.588,A -85,B 0,C 180,E1 -5586.329,E2 -5586.329} C_VEL
LIN {X 0,Y 509.917,Z 256.594,A -85,B 0,C 180,E1 -5588.719,E2 -5588.719} C_VEL
LIN {X 0,Y 509.907,Z 256.597,A -85,B 0,C 180,E1 -5591.931,E2 -5591.931} C_VEL
LIN {X 0,Y 509.896,Z 256.595,A -85,B 0,C 180,E1 -5595.241,E2 -5595.241} C_VEL
LIN {X 0,Y 509.89,Z 256.6,A -85,B 0,C 180,E1 -5598,E2 -5598} C_VEL
LIN {X 0,Y 509.851,Z 256.602,A -85,B 0,C 180,E1 -5601,E2 -5601} C_VEL
LIN {X 0,Y 509.87,Z 256.601,A -85,B 0,C 180,E1 -5604.425,E2 -5604.425} C_VEL
LIN {X 0,Y 509.885,Z 256.597,A -85,B 0,C 180,E1 -5607.054,E2 -5607.054} C_VEL
LIN {X 0,Y 509.856,Z 256.603,A -85,B 0,C 180,E1 -5609.75,E2 -5609.75} C_VEL
LIN {X 0,Y 509.873,Z 256.599,A -85,B 0,C 180,E1 -5612.773,E2 -5612.773} C_VEL
LIN {X 0,Y 509.84,Z 256.604,A -85,B 0,C 180,E1 -5615.58,E2 -5615.58} C_VEL
LIN {X 0,Y 509.848,Z 256.603,A -85,B 0,C 180,E1 -5618.337,E2 -5618.337} C_VEL
LIN {X 0,Y 509.855,Z 256.602,A -85,B 0,C 180,E1 -5621.424,E2 -5621.424} C_VEL
LIN {X 0,Y 509.852,Z 256.601,A -85,B 0,C 180,E1 -5624.667,E2 -5624.667} C_VEL
LIN {X 0,Y 509.876,Z 256.601,A -85,B 0,C 180,E1 -5628.099,E2 -5628.099} C_VEL
LIN {X 0,Y 509.854,Z 256.601,A -85,B 0,C 180,E1 -5630.648,E2 -5630.648} C_VEL
LIN {X 0,Y 509.826,Z 256.607,A -85,B 0,C 180,E1 -5633.733,E2 -5633.733} C_VEL
LIN {X 0,Y 509.159,Z 256.689,A -85,B 0,C 180,E1 -5634.393,E2 -5634.393} C_VEL
LIN {X 0,Y 506.341,Z 257.041,A -85,B 0,C 180,E1 -5635.465,E2 -5635.465} C_VEL
LIN {X 0,Y 503.948,Z 257.339,A -85,B 0,C 180,E1 -5636.328,E2 -5636.328} C_VEL
LIN {X 0,Y 502.9,Z 257.469,A -85,B 0,C 180,E1 -5636.995,E2 -5636.995} C_VEL
LIN {X 0,Y 502.802,Z 257.479,A -85,B 0,C 180,E1 -5637.22,E2 -5637.22} C_VEL
LIN {X 0,Y 502.823,Z 257.478,A -85,B 0,C 180,E1 -5640.061,E2 -5640.061} C_VEL
LIN {X 0,Y 502.828,Z 257.476,A -85,B 0,C 180,E1 -5642.532,E2 -5642.532} C_VEL
LIN {X 0,Y 502.82,Z 257.479,A -85,B 0,C 180,E1 -5645.297,E2 -5645.297} C_VEL
LIN {X 0,Y 502.785,Z 257.484,A -85,B 0,C 180,E1 -5647.826,E2 -5647.826} C_VEL
LIN {X 0,Y 502.816,Z 257.478,A -85,B 0,C 180,E1 -5650.399,E2 -5650.399} C_VEL
LIN {X 0,Y 502.827,Z 257.477,A -85,B 0,C 180,E1 -5652.931,E2 -5652.931} C_VEL
LIN {X 0,Y 502.842,Z 257.478,A -85,B 0,C 180,E1 -5655.429,E2 -5655.429} C_VEL
LIN {X 0,Y 502.885,Z 257.47,A -85,B 0,C 180,E1 -5658.716,E2 -5658.716} C_VEL
LIN {X 0,Y 502.892,Z 257.468,A -85,B 0,C 180,E1 -5661.966,E2 -5661.966} C_VEL
LIN {X 0,Y 502.903,Z 257.466,A -85,B 0,C 180,E1 -5664.386,E2 -5664.386} C_VEL
LIN {X 0,Y 502.489,Z 257.522,A -85,B 0,C 180,E1 -5667.595,E2 -5667.595} C_VEL
LIN {X 0,Y 502.757,Z 258.774,A -85,B 0,C 180,E1 -5669.198,E2 -5669.198} C_VEL
LIN {X 0,Y 502.405,Z 261.1,A -85,B 0,C 180,E1 -5671.603,E2 -5671.603} C_VEL
LIN {X 0,Y 502.411,Z 264.125,A -85,B 0,C 180,E1 -5674.814,E2 -5674.814} C_VEL
LIN {X 0,Y 502.354,Z 266.434,A -85,B 0,C 180,E1 -5677.233,E2 -5677.233} C_VEL
LIN {X 0,Y 502.272,Z 269.543,A -85,B 0,C 180,E1 -5680.48,E2 -5680.48} C_VEL
LIN {X 0,Y 502.258,Z 271.866,A -85,B 0,C 180,E1 -5682.885,E2 -5682.885} C_VEL
LIN {X 0,Y 506.658,Z 286.937,A -85,B 0,C 180,E1 -5683.409,E2 -5683.409} C_VEL
LIN {X 0,Y 507.264,Z 289.911,A -85,B 0,C 180,E1 -5683.52,E2 -5683.52} C_VEL
LIN {X 0,Y 506.888,Z 304.331,A -85,B 0,C 180,E1 -5684.001,E2 -5684.001} C_VEL
LIN {X 0,Y 506.393,Z 318.282,A -85,B 0,C 180,E1 -5684.62,E2 -5684.62} C_VEL
LIN {X 0,Y 505.923,Z 330.568,A -85,B 0,C 180,E1 -5685.303,E2 -5685.303} C_VEL
LIN {X 0,Y 505.3,Z 344.614,A -85,B 0,C 180,E1 -5686.271,E2 -5686.271} C_VEL
LIN {X 0,Y 504.769,Z 356.994,A -85,B 0,C 180,E1 -5687.313,E2 -5687.313} C_VEL
LIN {X 0,Y 504.087,Z 369.219,A -85,B 0,C 180,E1 -5688.553,E2 -5688.553} C_VEL
LIN {X 0,Y 503.596,Z 379.351,A -85,B 0,C 180,E1 -5689.78,E2 -5689.78} C_VEL
LIN {X 0,Y 503.138,Z 388.609,A -85,B 0,C 180,E1 -5691.116,E2 -5691.116} C_VEL
LIN {X 0,Y 502.824,Z 396.282,A -85,B 0,C 180,E1 -5692.434,E2 -5692.434} C_VEL
LIN {X 0,Y 502.535,Z 403.545,A -85,B 0,C 180,E1 -5693.926,E2 -5693.926} C_VEL
LIN {X 0,Y 502.371,Z 408.914,A -85,B 0,C 180,E1 -5695.257,E2 -5695.257} C_VEL
LIN {X 0,Y 502.241,Z 413.309,A -85,B 0,C 180,E1 -5696.601,E2 -5696.601} C_VEL
LIN {X 0,Y 502.098,Z 417.231,A -85,B 0,C 180,E1 -5698.14,E2 -5698.14} C_VEL
LIN {X 0,Y 502.049,Z 420.202,A -85,B 0,C 180,E1 -5699.786,E2 -5699.786} C_VEL
LIN {X 0,Y 501.997,Z 421.925,A -85,B 0,C 180,E1 -5701.353,E2 -5701.353} C_VEL
LIN {X 0,Y 501.988,Z 422.565,A -85,B 0,C 180,E1 -5703.093,E2 -5703.093} C_VEL
LIN {X 0,Y 502.013,Z 422.186,A -85,B 0,C 180,E1 -5704.315,E2 -5704.315} C_VEL
LIN {X 0,Y 501.984,Z 420.637,A -85,B 0,C 180,E1 -5706.016,E2 -5706.016} C_VEL
LIN {X 0,Y 502.049,Z 419.017,A -85,B 0,C 180,E1 -5707.07,E2 -5707.07} C_VEL
LIN {X 0,Y 502.188,Z 416.289,A -85,B 0,C 180,E1 -5708.401,E2 -5708.401} C_VEL
LIN {X 0,Y 502.301,Z 411.647,A -85,B 0,C 180,E1 -5710.061,E2 -5710.061} C_VEL
LIN {X 0,Y 502.445,Z 405.912,A -85,B 0,C 180,E1 -5711.636,E2 -5711.636} C_VEL
LIN {X 0,Y 502.716,Z 398.626,A -85,B 0,C 180,E1 -5713.236,E2 -5713.236} C_VEL
LIN {X 0,Y 503.141,Z 390.328,A -85,B 0,C 180,E1 -5714.719,E2 -5714.719} C_VEL
LIN {X 0,Y 503.537,Z 381.151,A -85,B 0,C 180,E1 -5716.086,E2 -5716.086} C_VEL
LIN {X 0,Y 504.06,Z 370.408,A -85,B 0,C 180,E1 -5717.424,E2 -5717.424} C_VEL
LIN {X 0,Y 504.677,Z 358.651,A -85,B 0,C 180,E1 -5718.641,E2 -5718.641} C_VEL
LIN {X 0,Y 505.318,Z 346.583,A -85,B 0,C 180,E1 -5719.679,E2 -5719.679} C_VEL
LIN {X 0,Y 505.832,Z 333.977,A -85,B 0,C 180,E1 -5720.584,E2 -5720.584} C_VEL
LIN {X 0,Y 506.413,Z 320.733,A -85,B 0,C 180,E1 -5721.355,E2 -5721.355} C_VEL
LIN {X 0,Y 506.848,Z 306.61,A -85,B 0,C 180,E1 -5722.01,E2 -5722.01} C_VEL
LIN {X 0,Y 507.264,Z 291.072,A -85,B 0,C 180,E1 -5722.545,E2 -5722.545} C_VEL
LIN {X 0,Y 507.061,Z 288.387,A -85,B 0,C 180,E1 -5722.632,E2 -5722.632} C_VEL
LIN {X 0,Y 504.237,Z 278.748,A -85,B 0,C 180,E1 -5722.984,E2 -5722.984} C_VEL
LIN {X 0,Y 502.295,Z 272.432,A -85,B 0,C 180,E1 -5723.202,E2 -5723.202} C_VEL
LIN {X 0,Y 502.303,Z 269.891,A -85,B 0,C 180,E1 -5725.969,E2 -5725.969} C_VEL
LIN {X 0,Y 502.409,Z 267.297,A -85,B 0,C 180,E1 -5728.831,E2 -5728.831} C_VEL
LIN {X 0,Y 502.454,Z 264.621,A -85,B 0,C 180,E1 -5731.786,E2 -5731.786} C_VEL
LIN {X 0,Y 502.481,Z 262.352,A -85,B 0,C 180,E1 -5734.306,E2 -5734.306} C_VEL
LIN {X 0,Y 502.557,Z 259.559,A -85,B 0,C 180,E1 -5737.363,E2 -5737.363} C_VEL
LIN {X 0,Y 502.578,Z 257.571,A -85,B 0,C 180,E1 -5739.539,E2 -5739.539} C_VEL
LIN {X 0,Y 502.774,Z 257.486,A -85,B 0,C 180,E1 -5742.091,E2 -5742.091} C_VEL
LIN {X 0,Y 502.832,Z 257.479,A -85,B 0,C 180,E1 -5744.663,E2 -5744.663} C_VEL
LIN {X 0,Y 502.87,Z 257.472,A -85,B 0,C 180,E1 -5748.04,E2 -5748.04} C_VEL
LIN {X 0,Y 502.87,Z 257.473,A -85,B 0,C 180,E1 -5751.158,E2 -5751.158} C_VEL
LIN {X 0,Y 502.924,Z 257.466,A -85,B 0,C 180,E1 -5753.582,E2 -5753.582} C_VEL
LIN {X 0,Y 502.896,Z 257.469,A -85,B 0,C 180,E1 -5756.796,E2 -5756.796} C_VEL
LIN {X 0,Y 503.031,Z 257.454,A -85,B 0,C 180,E1 -5759.2,E2 -5759.2} C_VEL
LIN {X 0,Y 502.898,Z 257.468,A -85,B 0,C 180,E1 -5761.602,E2 -5761.602} C_VEL
LIN {X 0,Y 502.897,Z 257.469,A -85,B 0,C 180,E1 -5763.205,E2 -5763.205} C_VEL
LIN {X 0,Y 502.925,Z 257.464,A -85,B 0,C 180,E1 -5766.42,E2 -5766.42} C_VEL
LIN {X 0,Y 502.872,Z 257.472,A -85,B 0,C 180,E1 -5768.844,E2 -5768.844} C_VEL
LIN {X 0,Y 502.843,Z 257.476,A -85,B 0,C 180,E1 -5772.102,E2 -5772.102} C_VEL
LIN {X 0,Y 502.845,Z 257.475,A -85,B 0,C 180,E1 -5775.4,E2 -5775.4} C_VEL
LIN {X 0,Y 502.843,Z 257.476,A -85,B 0,C 180,E1 -5778.123,E2 -5778.123} C_VEL
LIN {X 0,Y 502.826,Z 257.479,A -85,B 0,C 180,E1 -5780.537,E2 -5780.537} C_VEL
LIN {X 0,Y 502.795,Z 257.481,A -85,B 0,C 180,E1 -5783.041,E2 -5783.041} C_VEL
LIN {X 0,Y 502.84,Z 257.476,A -85,B 0,C 180,E1 -5785.676,E2 -5785.676} C_VEL
LIN {X 0,Y 502.838,Z 257.477,A -85,B 0,C 180,E1 -5788.373,E2 -5788.373} C_VEL
LIN {X 0,Y 502.79,Z 257.485,A -85,B 0,C 180,E1 -5791.499,E2 -5791.499} C_VEL
LIN {X 0,Y 502.801,Z 257.485,A -85,B 0,C 180,E1 -5793.995,E2 -5793.995} C_VEL
LIN {X 0,Y 502.776,Z 257.488,A -85,B 0,C 180,E1 -5797.179,E2 -5797.179} C_VEL
LIN {X 0,Y 502.786,Z 257.485,A -85,B 0,C 180,E1 -5800.016,E2 -5800.016} C_VEL
LIN {X 0,Y 502.801,Z 257.482,A -85,B 0,C 180,E1 -5802.2,E2 -5802.2} C_VEL
LIN {X 0,Y 502.839,Z 257.684,A -85,B 0,C 180,E1 -5803.945,E2 -5803.945} C_VEL
LIN {X 0,Y 503.948,Z 263.552,A -85,B 0,C 180,E1 -5806.895,E2 -5806.895} C_VEL
LIN {X 0,Y 504.343,Z 268.629,A -85,B 0,C 180,E1 -5809.086,E2 -5809.086} C_VEL
LIN {X 0,Y 504.135,Z 275.035,A -85,B 0,C 180,E1 -5811.741,E2 -5811.741} C_VEL
LIN {X 0,Y 503.823,Z 282.443,A -85,B 0,C 180,E1 -5814.628,E2 -5814.628} C_VEL
LIN {X 0,Y 503.61,Z 290.186,A -85,B 0,C 180,E1 -5817.502,E2 -5817.502} C_VEL
LIN {X 0,Y 503.429,Z 298.203,A -85,B 0,C 180,E1 -5820.347,E2 -5820.347} C_VEL
LIN {X 0,Y 503.236,Z 307.345,A -85,B 0,C 180,E1 -5823.456,E2 -5823.456} C_VEL
LIN {X 0,Y 502.988,Z 316.01,A -85,B 0,C 180,E1 -5826.534,E2 -5826.534} C_VEL
LIN {X 0,Y 502.758,Z 325.124,A -85,B 0,C 180,E1 -5829.701,E2 -5829.701} C_VEL
LIN {X 0,Y 502.735,Z 325.419,A -85,B 0,C 180,E1 -5829.802,E2 -5829.802} C_VEL
LIN {X 0,Y 506.913,Z 342.28,A -85,B 0,C 180,E1 -5830.301,E2 -5830.301} C_VEL
LIN {X 0,Y 507.295,Z 345.193,A -85,B 0,C 180,E1 -5830.391,E2 -5830.391} C_VEL
LIN {X 0,Y 506.909,Z 359.594,A -85,B 0,C 180,E1 -5830.839,E2 -5830.839} C_VEL
LIN {X 0,Y 506.381,Z 374.838,A -85,B 0,C 180,E1 -5831.49,E2 -5831.49} C_VEL
LIN {X 0,Y 505.822,Z 387.893,A -85,B 0,C 180,E1 -5832.202,E2 -5832.202} C_VEL
LIN {X 0,Y 505.21,Z 401.469,A -85,B 0,C 180,E1 -5833.119,E2 -5833.119} C_VEL
LIN {X 0,Y 504.62,Z 414.63,A -85,B 0,C 180,E1 -5834.206,E2 -5834.206} C_VEL
LIN {X 0,Y 504.044,Z 425.286,A -85,B 0,C 180,E1 -5835.259,E2 -5835.259} C_VEL
LIN {X 0,Y 503.55,Z 435.77,A -85,B 0,C 180,E1 -5836.481,E2 -5836.481} C_VEL
LIN {X 0,Y 503.006,Z 446.021,A -85,B 0,C 180,E1 -5837.903,E2 -5837.903} C_VEL
LIN {X 0,Y 502.794,Z 454.536,A -85,B 0,C 180,E1 -5839.327,E2 -5839.327} C_VEL
LIN {X 0,Y 502.467,Z 461.618,A -85,B 0,C 180,E1 -5840.744,E2 -5840.744} C_VEL
LIN {X 0,Y 502.296,Z 468.186,A -85,B 0,C 180,E1 -5842.362,E2 -5842.362} C_VEL
LIN {X 0,Y 502.198,Z 473.323,A -85,B 0,C 180,E1 -5843.976,E2 -5843.976} C_VEL
LIN {X 0,Y 502.082,Z 476.293,A -85,B 0,C 180,E1 -5845.183,E2 -5845.183} C_VEL
LIN {X 0,Y 502.107,Z 479.186,A -85,B 0,C 180,E1 -5846.791,E2 -5846.791} C_VEL
LIN {X 0,Y 502.033,Z 480.91,A -85,B 0,C 180,E1 -5848.396,E2 -5848.396} C_VEL
LIN {X 0,Y 501.977,Z 481.5,A -85,B 0,C 180,E1 -5850.001,E2 -5850.001} C_VEL
LIN {X 0,Y 502.033,Z 480.908,A -85,B 0,C 180,E1 -5851.605,E2 -5851.605} C_VEL
LIN {X 0,Y 502.107,Z 479.181,A -85,B 0,C 180,E1 -5853.21,E2 -5853.21} C_VEL
LIN {X 0,Y 502.082,Z 476.288,A -85,B 0,C 180,E1 -5854.818,E2 -5854.818} C_VEL
LIN {X 0,Y 502.187,Z 472.038,A -85,B 0,C 180,E1 -5856.47,E2 -5856.47} C_VEL
LIN {X 0,Y 502.325,Z 466.699,A -85,B 0,C 180,E1 -5858.043,E2 -5858.043} C_VEL
LIN {X 0,Y 502.491,Z 459.743,A -85,B 0,C 180,E1 -5859.663,E2 -5859.663} C_VEL
LIN {X 0,Y 502.887,Z 452.289,A -85,B 0,C 180,E1 -5861.079,E2 -5861.079} C_VEL
LIN {X 0,Y 503.176,Z 443.303,A -85,B 0,C 180,E1 -5862.504,E2 -5862.504} C_VEL
LIN {X 0,Y 503.697,Z 432.504,A -85,B 0,C 180,E1 -5863.928,E2 -5863.928} C_VEL
LIN {X 0,Y 504.248,Z 420.351,A -85,B 0,C 180,E1 -5865.253,E2 -5865.253} C_VEL
LIN {X 0,Y 504.901,Z 407.955,A -85,B 0,C 180,E1 -5866.372,E2 -5866.372} C_VEL
LIN {X 0,Y 505.521,Z 394.24,A -85,B 0,C 180,E1 -5867.392,E2 -5867.392} C_VEL
LIN {X 0,Y 506.134,Z 380.76,A -85,B 0,C 180,E1 -5868.206,E2 -5868.206} C_VEL
LIN {X 0,Y 506.734,Z 366.578,A -85,B 0,C 180,E1 -5868.885,E2 -5868.885} C_VEL
LIN {X 0,Y 507.13,Z 351.701,A -85,B 0,C 180,E1 -5869.427,E2 -5869.427} C_VEL
LIN {X 0,Y 507.152,Z 343.382,A -85,B 0,C 180,E1 -5869.664,E2 -5869.664} C_VEL
LIN {X 0,Y 503.135,Z 327.296,A -85,B 0,C 180,E1 -5870.15,E2 -5870.15} C_VEL
LIN {X 0,Y 502.738,Z 325.361,A -85,B 0,C 180,E1 -5870.218,E2 -5870.218} C_VEL
LIN {X 0,Y 502.941,Z 317.244,A -85,B 0,C 180,E1 -5873.034,E2 -5873.034} C_VEL
LIN {X 0,Y 503.203,Z 308.579,A -85,B 0,C 180,E1 -5876.101,E2 -5876.101} C_VEL
LIN {X 0,Y 503.456,Z 299.505,A -85,B 0,C 180,E1 -5879.248,E2 -5879.248} C_VEL
LIN {X 0,Y 503.631,Z 291.679,A -85,B 0,C 180,E1 -5882.025,E2 -5882.025} C_VEL
LIN {X 0,Y 503.867,Z 284.151,A -85,B 0,C 180,E1 -5884.881,E2 -5884.881} C_VEL
LIN {X 0,Y 504.19,Z 276.584,A -85,B 0,C 180,E1 -5887.831,E2 -5887.831} C_VEL
LIN {X 0,Y 504.382,Z 270.288,A -85,B 0,C 180,E1 -5890.393,E2 -5890.393} C_VEL
LIN {X 0,Y 504.254,Z 265.678,A -85,B 0,C 180,E1 -5892.38,E2 -5892.38} C_VEL
LIN {X 0,Y 503.436,Z 260.889,A -85,B 0,C 180,E1 -5894.605,E2 -5894.605} C_VEL
LIN {X 0,Y 502.815,Z 257.478,A -85,B 0,C 180,E1 -5896.31,E2 -5896.31} C_VEL
LIN {X 0,Y 502.823,Z 257.479,A -85,B 0,C 180,E1 -5899.005,E2 -5899.005} C_VEL
LIN {X 0,Y 502.798,Z 257.481,A -85,B 0,C 180,E1 -5902.046,E2 -5902.046} C_VEL
LIN {X 0,Y 502.801,Z 257.481,A -85,B 0,C 180,E1 -5905.034,E2 -5905.034} C_VEL
LIN {X 0,Y 502.788,Z 257.484,A -85,B 0,C 180,E1 -5907.915,E2 -5907.915} C_VEL
LIN {X 0,Y 502.828,Z 257.478,A -85,B 0,C 180,E1 -5910.712,E2 -5910.712} C_VEL
LIN {X 0,Y 502.869,Z 257.471,A -85,B 0,C 180,E1 -5913.439,E2 -5913.439} C_VEL
LIN {X 0,Y 502.791,Z 257.481,A -85,B 0,C 180,E1 -5916.086,E2 -5916.086} C_VEL
LIN {X 0,Y 502.789,Z 257.483,A -85,B 0,C 180,E1 -5918.688,E2 -5918.688} C_VEL
LIN {X 0,Y 502.836,Z 257.477,A -85,B 0,C 180,E1 -5921.248,E2 -5921.248} C_VEL
LIN {X 0,Y 502.828,Z 257.477,A -85,B 0,C 180,E1 -5923.767,E2 -5923.767} C_VEL
LIN {X 0,Y 502.835,Z 257.477,A -85,B 0,C 180,E1 -5926.254,E2 -5926.254} C_VEL
LIN {X 0,Y 502.882,Z 257.472,A -85,B 0,C 180,E1 -5928.716,E2 -5928.716} C_VEL
LIN {X 0,Y 502.906,Z 257.468,A -85,B 0,C 180,E1 -5931.966,E2 -5931.966} C_VEL
LIN {X 0,Y 502.931,Z 257.465,A -85,B 0,C 180,E1 -5934.386,E2 -5934.386} C_VEL
LIN {X 0,Y 503.029,Z 257.451,A -85,B 0,C 180,E1 -5937.597,E2 -5937.597} C_VEL
LIN {X 0,Y 503.031,Z 257.452,A -85,B 0,C 180,E1 -5939.999,E2 -5939.999} C_VEL
LIN {X 0,Y 503.027,Z 257.454,A -85,B 0,C 180,E1 -5942.401,E2 -5942.401} C_VEL
LIN {X 0,Y 502.931,Z 257.467,A -85,B 0,C 180,E1 -5946.418,E2 -5946.418} C_VEL
LIN {X 0,Y 502.875,Z 257.471,A -85,B 0,C 180,E1 -5948.842,E2 -5948.842} C_VEL
LIN {X 0,Y 502.849,Z 257.475,A -85,B 0,C 180,E1 -5952.101,E2 -5952.101} C_VEL
LIN {X 0,Y 502.851,Z 257.473,A -85,B 0,C 180,E1 -5955.399,E2 -5955.399} C_VEL
LIN {X 0,Y 502.848,Z 257.476,A -85,B 0,C 180,E1 -5958.121,E2 -5958.121} C_VEL
LIN {X 0,Y 502.83,Z 257.477,A -85,B 0,C 180,E1 -5960.535,E2 -5960.535} C_VEL
LIN {X 0,Y 502.795,Z 257.481,A -85,B 0,C 180,E1 -5963.039,E2 -5963.039} C_VEL
LIN {X 0,Y 502.84,Z 257.476,A -85,B 0,C 180,E1 -5965.674,E2 -5965.674} C_VEL
LIN {X 0,Y 502.84,Z 257.477,A -85,B 0,C 180,E1 -5968.371,E2 -5968.371} C_VEL
LIN {X 0,Y 502.792,Z 257.482,A -85,B 0,C 180,E1 -5971.498,E2 -5971.498} C_VEL
LIN {X 0,Y 502.804,Z 257.481,A -85,B 0,C 180,E1 -5974.443,E2 -5974.443} C_VEL
LIN {X 0,Y 502.778,Z 257.483,A -85,B 0,C 180,E1 -5977.177,E2 -5977.177} C_VEL
LIN {X 0,Y 502.785,Z 257.484,A -85,B 0,C 180,E1 -5980.014,E2 -5980.014} C_VEL
LIN {X 0,Y 502.799,Z 257.481,A -85,B 0,C 180,E1 -5982.198,E2 -5982.198} C_VEL
LIN {X 0,Y 502.796,Z 257.482,A -85,B 0,C 180,E1 -5985.467,E2 -5985.467} C_VEL
LIN {X 0,Y 502.83,Z 257.478,A -85,B 0,C 180,E1 -5987.864,E2 -5987.864} C_VEL
LIN {X 0,Y 502.804,Z 257.479,A -85,B 0,C 180,E1 -5991.024,E2 -5991.024} C_VEL
LIN {X 0,Y 502.779,Z 257.484,A -85,B 0,C 180,E1 -5994.166,E2 -5994.166} C_VEL
LIN {X 0,Y 502.802,Z 257.479,A -85,B 0,C 180,E1 -5997.22,E2 -5997.22} C_VEL
LIN {X 0,Y 502.104,Z 257.568,A -85,B 0,C 180,E1 -5997.889,E2 -5997.889} C_VEL
LIN {X 0,Y 499.246,Z 257.924,A -85,B 0,C 180,E1 -5998.975,E2 -5998.975} C_VEL
LIN {X 0,Y 496.854,Z 258.223,A -85,B 0,C 180,E1 -5999.85,E2 -5999.85} C_VEL
LIN {X 0,Y 495.836,Z 258.347,A -85,B 0,C 180,E1 -6000.526,E2 -6000.526} C_VEL
LIN {X 0,Y 495.757,Z 258.356,A -85,B 0,C 180,E1 -6000.754,E2 -6000.754} C_VEL
LIN {X 0,Y 495.791,Z 258.355,A -85,B 0,C 180,E1 -6003.932,E2 -6003.932} C_VEL
LIN {X 0,Y 495.749,Z 258.36,A -85,B 0,C 180,E1 -6007.139,E2 -6007.139} C_VEL
LIN {X 0,Y 495.769,Z 258.357,A -85,B 0,C 180,E1 -6010.109,E2 -6010.109} C_VEL
LIN {X 0,Y 495.778,Z 258.355,A -85,B 0,C 180,E1 -6012.681,E2 -6012.681} C_VEL
LIN {X 0,Y 495.784,Z 258.355,A -85,B 0,C 180,E1 -6015.216,E2 -6015.216} C_VEL
LIN {X 0,Y 495.859,Z 258.345,A -85,B 0,C 180,E1 -6018.554,E2 -6018.554} C_VEL
LIN {X 0,Y 495.864,Z 258.344,A -85,B 0,C 180,E1 -6021.851,E2 -6021.851} C_VEL
LIN {X 0,Y 495.865,Z 258.342,A -85,B 0,C 180,E1 -6024.306,E2 -6024.306} C_VEL
LIN {X 0,Y 495.444,Z 258.4,A -85,B 0,C 180,E1 -6027.56,E2 -6027.56} C_VEL
LIN {X 0,Y 495.595,Z 258.749,A -85,B 0,C 180,E1 -6028.374,E2 -6028.374} C_VEL
LIN {X 0,Y 495.673,Z 260.268,A -85,B 0,C 180,E1 -6029.999,E2 -6029.999} C_VEL
LIN {X 0,Y 495.406,Z 264.126,A -85,B 0,C 180,E1 -6034.067,E2 -6034.067} C_VEL
LIN {X 0,Y 495.291,Z 267.234,A -85,B 0,C 180,E1 -6037.336,E2 -6037.336} C_VEL
LIN {X 0,Y 495.211,Z 270.379,A -85,B 0,C 180,E1 -6040.631,E2 -6040.631} C_VEL
LIN {X 0,Y 495.229,Z 272.268,A -85,B 0,C 180,E1 -6042.602,E2 -6042.602} C_VEL
LIN {X 0,Y 500.108,Z 288.815,A -85,B 0,C 180,E1 -6043.187,E2 -6043.187} C_VEL
LIN {X 0,Y 500.594,Z 291.32,A -85,B 0,C 180,E1 -6043.282,E2 -6043.282} C_VEL
LIN {X 0,Y 500.122,Z 305.84,A -85,B 0,C 180,E1 -6043.782,E2 -6043.782} C_VEL
LIN {X 0,Y 499.654,Z 319.021,A -85,B 0,C 180,E1 -6044.384,E2 -6044.384} C_VEL
LIN {X 0,Y 499.146,Z 331.58,A -85,B 0,C 180,E1 -6045.098,E2 -6045.098} C_VEL
LIN {X 0,Y 498.551,Z 343.941,A -85,B 0,C 180,E1 -6045.955,E2 -6045.955} C_VEL
LIN {X 0,Y 497.922,Z 356.487,A -85,B 0,C 180,E1 -6047.009,E2 -6047.009} C_VEL
LIN {X 0,Y 497.234,Z 368.862,A -85,B 0,C 180,E1 -6048.262,E2 -6048.262} C_VEL
LIN {X 0,Y 496.648,Z 380.085,A -85,B 0,C 180,E1 -6049.638,E2 -6049.638} C_VEL
LIN {X 0,Y 496.186,Z 388.925,A -85,B 0,C 180,E1 -6050.933,E2 -6050.933} C_VEL
LIN {X 0,Y 495.801,Z 397.865,A -85,B 0,C 180,E1 -6052.502,E2 -6052.502} C_VEL
LIN {X 0,Y 495.516,Z 404.16,A -85,B 0,C 180,E1 -6053.842,E2 -6053.842} C_VEL
LIN {X 0,Y 495.327,Z 409.493,A -85,B 0,C 180,E1 -6055.192,E2 -6055.192} C_VEL
LIN {X 0,Y 495.19,Z 414.028,A -85,B 0,C 180,E1 -6056.607,E2 -6056.607} C_VEL
LIN {X 0,Y 495.013,Z 418.226,A -85,B 0,C 180,E1 -6058.331,E2 -6058.331} C_VEL
LIN {X 0,Y 494.962,Z 420.977,A -85,B 0,C 180,E1 -6059.99,E2 -6059.99} C_VEL
LIN {X 0,Y 494.928,Z 422.573,A -85,B 0,C 180,E1 -6061.694,E2 -6061.694} C_VEL
LIN {X 0,Y 494.929,Z 423.004,A -85,B 0,C 180,E1 -6063.094,E2 -6063.094} C_VEL
LIN {X 0,Y 494.937,Z 422.472,A -85,B 0,C 180,E1 -6064.609,E2 -6064.609} C_VEL
LIN {X 0,Y 494.901,Z 421.214,A -85,B 0,C 180,E1 -6065.961,E2 -6065.961} C_VEL
LIN {X 0,Y 495.033,Z 418.582,A -85,B 0,C 180,E1 -6067.623,E2 -6067.623} C_VEL
LIN {X 0,Y 495.162,Z 414.979,A -85,B 0,C 180,E1 -6069.167,E2 -6069.167} C_VEL
LIN {X 0,Y 495.3,Z 410.125,A -85,B 0,C 180,E1 -6070.745,E2 -6070.745} C_VEL
LIN {X 0,Y 495.507,Z 404.725,A -85,B 0,C 180,E1 -6072.15,E2 -6072.15} C_VEL
LIN {X 0,Y 495.817,Z 397.397,A -85,B 0,C 180,E1 -6073.707,E2 -6073.707} C_VEL
LIN {X 0,Y 496.209,Z 389.578,A -85,B 0,C 180,E1 -6075.085,E2 -6075.085} C_VEL
LIN {X 0,Y 496.671,Z 380.078,A -85,B 0,C 180,E1 -6076.484,E2 -6076.484} C_VEL
LIN {X 0,Y 497.331,Z 368.507,A -85,B 0,C 180,E1 -6077.892,E2 -6077.892} C_VEL
LIN {X 0,Y 497.945,Z 357.293,A -85,B 0,C 180,E1 -6079.033,E2 -6079.033} C_VEL
LIN {X 0,Y 498.694,Z 344.406,A -85,B 0,C 180,E1 -6080.119,E2 -6080.119} C_VEL
LIN {X 0,Y 499.209,Z 331.843,A -85,B 0,C 180,E1 -6080.996,E2 -6080.996} C_VEL
LIN {X 0,Y 499.843,Z 317.824,A -85,B 0,C 180,E1 -6081.783,E2 -6081.783} C_VEL
LIN {X 0,Y 500.323,Z 303.198,A -85,B 0,C 180,E1 -6082.425,E2 -6082.425} C_VEL
LIN {X 0,Y 500.472,Z 290.234,A -85,B 0,C 180,E1 -6082.856,E2 -6082.856} C_VEL
LIN {X 0,Y 498.201,Z 282.159,A -85,B 0,C 180,E1 -6083.165,E2 -6083.165} C_VEL
LIN {X 0,Y 495.223,Z 272.921,A -85,B 0,C 180,E1 -6083.503,E2 -6083.503} C_VEL
LIN {X 0,Y 495.262,Z 270.286,A -85,B 0,C 180,E1 -6086.399,E2 -6086.399} C_VEL
LIN {X 0,Y 495.344,Z 267.67,A -85,B 0,C 180,E1 -6089.286,E2 -6089.286} C_VEL
LIN {X 0,Y 495.391,Z 265.176,A -85,B 0,C 180,E1 -6092.086,E2 -6092.086} C_VEL
LIN {X 0,Y 495.465,Z 262.348,A -85,B 0,C 180,E1 -6095.204,E2 -6095.204} C_VEL
LIN {X 0,Y 495.524,Z 260.287,A -85,B 0,C 180,E1 -6097.485,E2 -6097.485} C_VEL
LIN {X 0,Y 495.538,Z 258.56,A -85,B 0,C 180,E1 -6099.396,E2 -6099.396} C_VEL
LIN {X 0,Y 495.724,Z 258.364,A -85,B 0,C 180,E1 -6101.827,E2 -6101.827} C_VEL
LIN {X 0,Y 495.816,Z 258.354,A -85,B 0,C 180,E1 -6104.549,E2 -6104.549} C_VEL
LIN {X 0,Y 495.822,Z 258.351,A -85,B 0,C 180,E1 -6107.966,E2 -6107.966} C_VEL
LIN {X 0,Y 495.838,Z 258.349,A -85,B 0,C 180,E1 -6111.031,E2 -6111.031} C_VEL
LIN {X 0,Y 495.875,Z 258.344,A -85,B 0,C 180,E1 -6113.491,E2 -6113.491} C_VEL
LIN {X 0,Y 495.841,Z 258.348,A -85,B 0,C 180,E1 -6116.751,E2 -6116.751} C_VEL
LIN {X 0,Y 496.001,Z 258.329,A -85,B 0,C 180,E1 -6119.189,E2 -6119.189} C_VEL
LIN {X 0,Y 495.868,Z 258.344,A -85,B 0,C 180,E1 -6121.625,E2 -6121.625} C_VEL
LIN {X 0,Y 495.841,Z 258.348,A -85,B 0,C 180,E1 -6123.251,E2 -6123.251} C_VEL
LIN {X 0,Y 495.876,Z 258.343,A -85,B 0,C 180,E1 -6126.511,E2 -6126.511} C_VEL
LIN {X 0,Y 495.841,Z 258.349,A -85,B 0,C 180,E1 -6128.971,E2 -6128.971} C_VEL
LIN {X 0,Y 495.825,Z 258.351,A -85,B 0,C 180,E1 -6132.036,E2 -6132.036} C_VEL
LIN {X 0,Y 495.821,Z 258.35,A -85,B 0,C 180,E1 -6135.453,E2 -6135.453} C_VEL
LIN {X 0,Y 495.804,Z 258.353,A -85,B 0,C 180,E1 -6138.248,E2 -6138.248} C_VEL
LIN {X 0,Y 495.771,Z 258.356,A -85,B 0,C 180,E1 -6140.757,E2 -6140.757} C_VEL
LIN {X 0,Y 495.75,Z 258.359,A -85,B 0,C 180,E1 -6143.388,E2 -6143.388} C_VEL
LIN {X 0,Y 495.797,Z 258.354,A -85,B 0,C 180,E1 -6146.068,E2 -6146.068} C_VEL
LIN {X 0,Y 495.77,Z 258.359,A -85,B 0,C 180,E1 -6148.815,E2 -6148.815} C_VEL
LIN {X 0,Y 495.753,Z 258.363,A -85,B 0,C 180,E1 -6151.726,E2 -6151.726} C_VEL
LIN {X 0,Y 495.767,Z 258.362,A -85,B 0,C 180,E1 -6154.695,E2 -6154.695} C_VEL
LIN {X 0,Y 495.728,Z 258.367,A -85,B 0,C 180,E1 -6157.562,E2 -6157.562} C_VEL
LIN {X 0,Y 495.765,Z 258.359,A -85,B 0,C 180,E1 -6160.701,E2 -6160.701} C_VEL
LIN {X 0,Y 495.741,Z 258.418,A -85,B 0,C 180,E1 -6163.506,E2 -6163.506} C_VEL
LIN {X 0,Y 496.969,Z 264.693,A -85,B 0,C 180,E1 -6166.716,E2 -6166.716} C_VEL
LIN {X 0,Y 497.335,Z 268.603,A -85,B 0,C 180,E1 -6168.501,E2 -6168.501} C_VEL
LIN {X 0,Y 497.23,Z 274.613,A -85,B 0,C 180,E1 -6171.022,E2 -6171.022} C_VEL
LIN {X 0,Y 496.925,Z 281.302,A -85,B 0,C 180,E1 -6173.722,E2 -6173.722} C_VEL
LIN {X 0,Y 496.644,Z 289.999,A -85,B 0,C 180,E1 -6177.037,E2 -6177.037} C_VEL
LIN {X 0,Y 496.382,Z 298.962,A -85,B 0,C 180,E1 -6180.295,E2 -6180.295} C_VEL
LIN {X 0,Y 496.202,Z 307.312,A -85,B 0,C 180,E1 -6183.165,E2 -6183.165} C_VEL
LIN {X 0,Y 496.003,Z 314.772,A -85,B 0,C 180,E1 -6185.739,E2 -6185.739} C_VEL
LIN {X 0,Y 495.786,Z 323.436,A -85,B 0,C 180,E1 -6188.81,E2 -6188.81} C_VEL
LIN {X 0,Y 495.723,Z 325.425,A -85,B 0,C 180,E1 -6189.505,E2 -6189.505} C_VEL
LIN {X 0,Y 499.881,Z 342.049,A -85,B 0,C 180,E1 -6190.007,E2 -6190.007} C_VEL
LIN {X 0,Y 500.578,Z 346.169,A -85,B 0,C 180,E1 -6190.146,E2 -6190.146} C_VEL
LIN {X 0,Y 500.155,Z 360.715,A -85,B 0,C 180,E1 -6190.616,E2 -6190.616} C_VEL
LIN {X 0,Y 499.652,Z 374.837,A -85,B 0,C 180,E1 -6191.232,E2 -6191.232} C_VEL
LIN {X 0,Y 499.034,Z 387.895,A -85,B 0,C 180,E1 -6191.952,E2 -6191.952} C_VEL
LIN {X 0,Y 498.382,Z 401.47,A -85,B 0,C 180,E1 -6192.881,E2 -6192.881} C_VEL
LIN {X 0,Y 497.766,Z 413.925,A -85,B 0,C 180,E1 -6193.919,E2 -6193.919} C_VEL
LIN {X 0,Y 497.138,Z 425.286,A -85,B 0,C 180,E1 -6195.049,E2 -6195.049} C_VEL
LIN {X 0,Y 496.609,Z 435.77,A -85,B 0,C 180,E1 -6196.288,E2 -6196.288} C_VEL
LIN {X 0,Y 496.033,Z 446.02,A -85,B 0,C 180,E1 -6197.73,E2 -6197.73} C_VEL
LIN {X 0,Y 495.755,Z 454.536,A -85,B 0,C 180,E1 -6199.174,E2 -6199.174} C_VEL
LIN {X 0,Y 495.407,Z 461.618,A -85,B 0,C 180,E1 -6200.611,E2 -6200.611} C_VEL
LIN {X 0,Y 495.211,Z 468.185,A -85,B 0,C 180,E1 -6202.252,E2 -6202.252} C_VEL
LIN {X 0,Y 495.108,Z 473.036,A -85,B 0,C 180,E1 -6203.779,E2 -6203.779} C_VEL
LIN {X 0,Y 495.007,Z 476.293,A -85,B 0,C 180,E1 -6205.114,E2 -6205.114} C_VEL
LIN {X 0,Y 495.027,Z 479.186,A -85,B 0,C 180,E1 -6206.745,E2 -6206.745} C_VEL
LIN {X 0,Y 494.959,Z 480.91,A -85,B 0,C 180,E1 -6208.373,E2 -6208.373} C_VEL
LIN {X 0,Y 494.895,Z 481.5,A -85,B 0,C 180,E1 -6210.001,E2 -6210.001} C_VEL
LIN {X 0,Y 494.959,Z 480.908,A -85,B 0,C 180,E1 -6211.628,E2 -6211.628} C_VEL
LIN {X 0,Y 495.027,Z 479.181,A -85,B 0,C 180,E1 -6213.256,E2 -6213.256} C_VEL
LIN {X 0,Y 495.007,Z 476.288,A -85,B 0,C 180,E1 -6214.887,E2 -6214.887} C_VEL
LIN {X 0,Y 495.123,Z 472.163,A -85,B 0,C 180,E1 -6216.521,E2 -6216.521} C_VEL
LIN {X 0,Y 495.254,Z 466.699,A -85,B 0,C 180,E1 -6218.159,E2 -6218.159} C_VEL
LIN {X 0,Y 495.438,Z 459.742,A -85,B 0,C 180,E1 -6219.801,E2 -6219.801} C_VEL
LIN {X 0,Y 495.871,Z 452.289,A -85,B 0,C 180,E1 -6221.238,E2 -6221.238} C_VEL
LIN {X 0,Y 496.183,Z 443.303,A -85,B 0,C 180,E1 -6222.683,E2 -6222.683} C_VEL
LIN {X 0,Y 496.766,Z 432.504,A -85,B 0,C 180,E1 -6224.126,E2 -6224.126} C_VEL
LIN {X 0,Y 497.363,Z 420.352,A -85,B 0,C 180,E1 -6225.469,E2 -6225.469} C_VEL
LIN {X 0,Y 498.063,Z 407.956,A -85,B 0,C 180,E1 -6226.604,E2 -6226.604} C_VEL
LIN {X 0,Y 498.736,Z 394.242,A -85,B 0,C 180,E1 -6227.637,E2 -6227.637} C_VEL
LIN {X 0,Y 499.348,Z 380.761,A -85,B 0,C 180,E1 -6228.462,E2 -6228.462} C_VEL
LIN {X 0,Y 499.997,Z 366.837,A -85,B 0,C 180,E1 -6229.138,E2 -6229.138} C_VEL
LIN {X 0,Y 500.465,Z 351.701,A -85,B 0,C 180,E1 -6229.697,E2 -6229.697} C_VEL
LIN {X 0,Y 500.475,Z 344.833,A -85,B 0,C 180,E1 -6229.898,E2 -6229.898} C_VEL
LIN {X 0,Y 496.834,Z 329.876,A -85,B 0,C 180,E1 -6230.374,E2 -6230.374} C_VEL
LIN {X 0,Y 495.724,Z 325.386,A -85,B 0,C 180,E1 -6230.509,E2 -6230.509} C_VEL
LIN {X 0,Y 495.927,Z 317.244,A -85,B 0,C 180,E1 -6233.379,E2 -6233.379} C_VEL
LIN {X 0,Y 496.166,Z 309.667,A -85,B 0,C 180,E1 -6236.047,E2 -6236.047} C_VEL
LIN {X 0,Y 496.426,Z 300.499,A -85,B 0,C 180,E1 -6239.238,E2 -6239.238} C_VEL
LIN {X 0,Y 496.583,Z 293.168,A -85,B 0,C 180,E1 -6241.879,E2 -6241.879} C_VEL
LIN {X 0,Y 496.855,Z 285.375,A -85,B 0,C 180,E1 -6244.874,E2 -6244.874} C_VEL
LIN {X 0,Y 497.186,Z 278.301,A -85,B 0,C 180,E1 -6247.665,E2 -6247.665} C_VEL
LIN {X 0,Y 497.428,Z 271.365,A -85,B 0,C 180,E1 -6250.536,E2 -6250.536} C_VEL
LIN {X 0,Y 497.361,Z 267.677,A -85,B 0,C 180,E1 -6252.142,E2 -6252.142} C_VEL
LIN {X 0,Y 496.58,Z 262.844,A -85,B 0,C 180,E1 -6254.411,E2 -6254.411} C_VEL
LIN {X 0,Y 495.734,Z 258.363,A -85,B 0,C 180,E1 -6256.694,E2 -6256.694} C_VEL
LIN {X 0,Y 495.771,Z 258.358,A -85,B 0,C 180,E1 -6259.3,E2 -6259.3} C_VEL
LIN {X 0,Y 495.734,Z 258.362,A -85,B 0,C 180,E1 -6262.438,E2 -6262.438} C_VEL
LIN {X 0,Y 495.776,Z 258.357,A -85,B 0,C 180,E1 -6265.456,E2 -6265.456} C_VEL
LIN {X 0,Y 495.76,Z 258.357,A -85,B 0,C 180,E1 -6268.364,E2 -6268.364} C_VEL
LIN {X 0,Y 495.791,Z 258.353,A -85,B 0,C 180,E1 -6271.507,E2 -6271.507} C_VEL
LIN {X 0,Y 495.796,Z 258.352,A -85,B 0,C 180,E1 -6273.932,E2 -6273.932} C_VEL
LIN {X 0,Y 495.766,Z 258.358,A -85,B 0,C 180,E1 -6277.139,E2 -6277.139} C_VEL
LIN {X 0,Y 495.778,Z 258.355,A -85,B 0,C 180,E1 -6280.109,E2 -6280.109} C_VEL
LIN {X 0,Y 495.792,Z 258.355,A -85,B 0,C 180,E1 -6282.681,E2 -6282.681} C_VEL
LIN {X 0,Y 495.795,Z 258.354,A -85,B 0,C 180,E1 -6285.217,E2 -6285.217} C_VEL
LIN {X 0,Y 495.857,Z 258.347,A -85,B 0,C 180,E1 -6288.554,E2 -6288.554} C_VEL
LIN {X 0,Y 495.877,Z 258.343,A -85,B 0,C 180,E1 -6291.851,E2 -6291.851} C_VEL
LIN {X 0,Y 495.842,Z 258.346,A -85,B 0,C 180,E1 -6295.121,E2 -6295.121} C_VEL
LIN {X 0,Y 495.998,Z 258.326,A -85,B 0,C 180,E1 -6297.563,E2 -6297.563} C_VEL
LIN {X 0,Y 496.002,Z 258.327,A -85,B 0,C 180,E1 -6299.999,E2 -6299.999} C_VEL
LIN {X 0,Y 495.995,Z 258.33,A -85,B 0,C 180,E1 -6302.435,E2 -6302.435} C_VEL
LIN {X 0,Y 495.898,Z 258.341,A -85,B 0,C 180,E1 -6305.693,E2 -6305.693} C_VEL
LIN {X 0,Y 495.876,Z 258.344,A -85,B 0,C 180,E1 -6308.147,E2 -6308.147} C_VEL
LIN {X 0,Y 495.854,Z 258.344,A -85,B 0,C 180,E1 -6311.444,E2 -6311.444} C_VEL
LIN {X 0,Y 495.792,Z 258.354,A -85,B 0,C 180,E1 -6314.782,E2 -6314.782} C_VEL
LIN {X 0,Y 495.788,Z 258.353,A -85,B 0,C 180,E1 -6317.317,E2 -6317.317} C_VEL
LIN {X 0,Y 495.772,Z 258.357,A -85,B 0,C 180,E1 -6319.889,E2 -6319.889} C_VEL
LIN {X 0,Y 495.762,Z 258.357,A -85,B 0,C 180,E1 -6322.86,E2 -6322.86} C_VEL
LIN {X 0,Y 495.791,Z 258.355,A -85,B 0,C 180,E1 -6326.067,E2 -6326.067} C_VEL
LIN {X 0,Y 495.771,Z 258.355,A -85,B 0,C 180,E1 -6328.813,E2 -6328.813} C_VEL
LIN {X 0,Y 495.754,Z 258.36,A -85,B 0,C 180,E1 -6331.724,E2 -6331.724} C_VEL
LIN {X 0,Y 495.774,Z 258.355,A -85,B 0,C 180,E1 -6334.694,E2 -6334.694} C_VEL
LIN {X 0,Y 495.728,Z 258.362,A -85,B 0,C 180,E1 -6337.56,E2 -6337.56} C_VEL
LIN {X 0,Y 495.763,Z 258.357,A -85,B 0,C 180,E1 -6340.698,E2 -6340.698} C_VEL
LIN {X 0,Y 495.73,Z 258.362,A -85,B 0,C 180,E1 -6343.694,E2 -6343.694} C_VEL
LIN {X 0,Y 495.73,Z 258.361,A -85,B 0,C 180,E1 -6346.303,E2 -6346.303} C_VEL
LIN {X 0,Y 495.774,Z 258.356,A -85,B 0,C 180,E1 -6349.3,E2 -6349.3} C_VEL
LIN {X 0,Y 495.726,Z 258.362,A -85,B 0,C 180,E1 -6352.437,E2 -6352.437} C_VEL
LIN {X 0,Y 495.778,Z 258.356,A -85,B 0,C 180,E1 -6355.456,E2 -6355.456} C_VEL
LIN {X 0,Y 495.752,Z 258.359,A -85,B 0,C 180,E1 -6358.363,E2 -6358.363} C_VEL
LIN {X 0,Y 495.757,Z 258.356,A -85,B 0,C 180,E1 -6360.754,E2 -6360.754} C_VEL
LIN {X 0,Y 495.096,Z 258.442,A -85,B 0,C 180,E1 -6361.433,E2 -6361.433} C_VEL
LIN {X 0,Y 492.239,Z 258.795,A -85,B 0,C 180,E1 -6362.536,E2 -6362.536} C_VEL
LIN {X 0,Y 489.83,Z 259.097,A -85,B 0,C 180,E1 -6363.424,E2 -6363.424} C_VEL
LIN {X 0,Y 488.812,Z 259.222,A -85,B 0,C 180,E1 -6364.111,E2 -6364.111} C_VEL
LIN {X 0,Y 488.738,Z 259.23,A -85,B 0,C 180,E1 -6364.343,E2 -6364.343} C_VEL
LIN {X 0,Y 488.712,Z 259.236,A -85,B 0,C 180,E1 -6367.152,E2 -6367.152} C_VEL
LIN {X 0,Y 488.72,Z 259.235,A -85,B 0,C 180,E1 -6369.81,E2 -6369.81} C_VEL
LIN {X 0,Y 488.725,Z 259.233,A -85,B 0,C 180,E1 -6372.423,E2 -6372.423} C_VEL
LIN {X 0,Y 488.755,Z 259.23,A -85,B 0,C 180,E1 -6374.999,E2 -6374.999} C_VEL
LIN {X 0,Y 488.821,Z 259.221,A -85,B 0,C 180,E1 -6378.387,E2 -6378.387} C_VEL
LIN {X 0,Y 488.809,Z 259.224,A -85,B 0,C 180,E1 -6381.733,E2 -6381.733} C_VEL
LIN {X 0,Y 488.827,Z 259.219,A -85,B 0,C 180,E1 -6384.223,E2 -6384.223} C_VEL
LIN {X 0,Y 488.448,Z 259.271,A -85,B 0,C 180,E1 -6386.7,E2 -6386.7} C_VEL
LIN {X 0,Y 488.527,Z 259.487,A -85,B 0,C 180,E1 -6388.351,E2 -6388.351} C_VEL
LIN {X 0,Y 488.615,Z 261.008,A -85,B 0,C 180,E1 -6389.999,E2 -6389.999} C_VEL
LIN {X 0,Y 488.361,Z 264.901,A -85,B 0,C 180,E1 -6394.126,E2 -6394.126} C_VEL
LIN {X 0,Y 488.223,Z 268.041,A -85,B 0,C 180,E1 -6397.443,E2 -6397.443} C_VEL
LIN {X 0,Y 488.159,Z 271.225,A -85,B 0,C 180,E1 -6400.786,E2 -6400.786} C_VEL
LIN {X 0,Y 488.165,Z 272.663,A -85,B 0,C 180,E1 -6402.289,E2 -6402.289} C_VEL
LIN {X 0,Y 493.382,Z 290.007,A -85,B 0,C 180,E1 -6402.931,E2 -6402.931} C_VEL
LIN {X 0,Y 493.881,Z 293.418,A -85,B 0,C 180,E1 -6403.055,E2 -6403.055} C_VEL
LIN {X 0,Y 493.389,Z 307.989,A -85,B 0,C 180,E1 -6403.585,E2 -6403.585} C_VEL
LIN {X 0,Y 492.848,Z 321.608,A -85,B 0,C 180,E1 -6404.239,E2 -6404.239} C_VEL
LIN {X 0,Y 492.25,Z 334.261,A -85,B 0,C 180,E1 -6404.997,E2 -6404.997} C_VEL
LIN {X 0,Y 491.619,Z 347.282,A -85,B 0,C 180,E1 -6405.952,E2 -6405.952} C_VEL
LIN {X 0,Y 490.968,Z 359.783,A -85,B 0,C 180,E1 -6407.064,E2 -6407.064} C_VEL
LIN {X 0,Y 490.293,Z 370.239,A -85,B 0,C 180,E1 -6408.165,E2 -6408.165} C_VEL
LIN {X 0,Y 489.701,Z 380.81,A -85,B 0,C 180,E1 -6409.491,E2 -6409.491} C_VEL
LIN {X 0,Y 489.154,Z 390.532,A -85,B 0,C 180,E1 -6410.953,E2 -6410.953} C_VEL
LIN {X 0,Y 488.787,Z 398.524,A -85,B 0,C 180,E1 -6412.397,E2 -6412.397} C_VEL
LIN {X 0,Y 488.501,Z 404.775,A -85,B 0,C 180,E1 -6413.755,E2 -6413.755} C_VEL
LIN {X 0,Y 488.257,Z 410.396,A -85,B 0,C 180,E1 -6415.22,E2 -6415.22} C_VEL
LIN {X 0,Y 488.129,Z 415.22,A -85,B 0,C 180,E1 -6416.793,E2 -6416.793} C_VEL
LIN {X 0,Y 487.934,Z 419.189,A -85,B 0,C 180,E1 -6418.527,E2 -6418.527} C_VEL
LIN {X 0,Y 487.872,Z 421.853,A -85,B 0,C 180,E1 -6420.277,E2 -6420.277} C_VEL
LIN {X 0,Y 487.836,Z 423.083,A -85,B 0,C 180,E1 -6421.793,E2 -6421.793} C_VEL
LIN {X 0,Y 487.831,Z 423.403,A -85,B 0,C 180,E1 -6423.326,E2 -6423.326} C_VEL
LIN {X 0,Y 487.825,Z 422.495,A -85,B 0,C 180,E1 -6425.188,E2 -6425.188} C_VEL
LIN {X 0,Y 487.838,Z 421.368,A -85,B 0,C 180,E1 -6426.222,E2 -6426.222} C_VEL
LIN {X 0,Y 487.952,Z 419.177,A -85,B 0,C 180,E1 -6427.614,E2 -6427.614} C_VEL
LIN {X 0,Y 488.115,Z 415.293,A -85,B 0,C 180,E1 -6429.31,E2 -6429.31} C_VEL
LIN {X 0,Y 488.252,Z 410.385,A -85,B 0,C 180,E1 -6430.914,E2 -6430.914} C_VEL
LIN {X 0,Y 488.539,Z 404.07,A -85,B 0,C 180,E1 -6432.541,E2 -6432.541} C_VEL
LIN {X 0,Y 488.9,Z 396.846,A -85,B 0,C 180,E1 -6434.05,E2 -6434.05} C_VEL
LIN {X 0,Y 489.328,Z 388.261,A -85,B 0,C 180,E1 -6435.535,E2 -6435.535} C_VEL
LIN {X 0,Y 489.92,Z 377.891,A -85,B 0,C 180,E1 -6437.02,E2 -6437.02} C_VEL
LIN {X 0,Y 490.596,Z 366.752,A -85,B 0,C 180,E1 -6438.342,E2 -6438.342} C_VEL
LIN {X 0,Y 491.256,Z 355.524,A -85,B 0,C 180,E1 -6439.459,E2 -6439.459} C_VEL
LIN {X 0,Y 491.968,Z 343.244,A -85,B 0,C 180,E1 -6440.48,E2 -6440.48} C_VEL
LIN {X 0,Y 492.532,Z 330.795,A -85,B 0,C 180,E1 -6441.342,E2 -6441.342} C_VEL
LIN {X 0,Y 493.172,Z 317.577,A -85,B 0,C 180,E1 -6442.082,E2 -6442.082} C_VEL
LIN {X 0,Y 493.668,Z 302.283,A -85,B 0,C 180,E1 -6442.749,E2 -6442.749} C_VEL
LIN {X 0,Y 493.812,Z 291.663,A -85,B 0,C 180,E1 -6443.104,E2 -6443.104} C_VEL
LIN {X 0,Y 491.16,Z 282.619,A -85,B 0,C 180,E1 -6443.465,E2 -6443.465} C_VEL
LIN {X 0,Y 488.175,Z 273.426,A -85,B 0,C 180,E1 -6443.796,E2 -6443.796} C_VEL
LIN {X 0,Y 488.244,Z 270.677,A -85,B 0,C 180,E1 -6446.841,E2 -6446.841} C_VEL
LIN {X 0,Y 488.286,Z 268.048,A -85,B 0,C 180,E1 -6449.752,E2 -6449.752} C_VEL
LIN {X 0,Y 488.334,Z 265.534,A -85,B 0,C 180,E1 -6452.58,E2 -6452.58} C_VEL
LIN {X 0,Y 488.421,Z 263.074,A -85,B 0,C 180,E1 -6455.338,E2 -6455.338} C_VEL
LIN {X 0,Y 488.45,Z 260.67,A -85,B 0,C 180,E1 -6458.033,E2 -6458.033} C_VEL
LIN {X 0,Y 488.52,Z 259.263,A -85,B 0,C 180,E1 -6459.803,E2 -6459.803} C_VEL
LIN {X 0,Y 488.682,Z 259.244,A -85,B 0,C 180,E1 -6462.423,E2 -6462.423} C_VEL
LIN {X 0,Y 488.755,Z 259.231,A -85,B 0,C 180,E1 -6465.001,E2 -6465.001} C_VEL
LIN {X 0,Y 488.799,Z 259.225,A -85,B 0,C 180,E1 -6468.388,E2 -6468.388} C_VEL
LIN {X 0,Y 488.812,Z 259.224,A -85,B 0,C 180,E1 -6471.735,E2 -6471.735} C_VEL
LIN {X 0,Y 488.851,Z 259.219,A -85,B 0,C 180,E1 -6474.225,E2 -6474.225} C_VEL
LIN {X 0,Y 488.958,Z 259.204,A -85,B 0,C 180,E1 -6477.53,E2 -6477.53} C_VEL
LIN {X 0,Y 488.951,Z 259.206,A -85,B 0,C 180,E1 -6480.824,E2 -6480.824} C_VEL
LIN {X 0,Y 488.957,Z 259.206,A -85,B 0,C 180,E1 -6482.472,E2 -6482.472} C_VEL
LIN {X 0,Y 488.853,Z 259.218,A -85,B 0,C 180,E1 -6485.777,E2 -6485.777} C_VEL
LIN {X 0,Y 488.815,Z 259.222,A -85,B 0,C 180,E1 -6488.267,E2 -6488.267} C_VEL
LIN {X 0,Y 488.802,Z 259.224,A -85,B 0,C 180,E1 -6491.613,E2 -6491.613} C_VEL
LIN {X 0,Y 488.759,Z 259.229,A -85,B 0,C 180,E1 -6495.001,E2 -6495.001} C_VEL
LIN {X 0,Y 488.752,Z 259.231,A -85,B 0,C 180,E1 -6498.443,E2 -6498.443} C_VEL
LIN {X 0,Y 488.705,Z 259.236,A -85,B 0,C 180,E1 -6501.071,E2 -6501.071} C_VEL
LIN {X 0,Y 488.692,Z 259.239,A -85,B 0,C 180,E1 -6503.746,E2 -6503.746} C_VEL
LIN {X 0,Y 488.797,Z 259.225,A -85,B 0,C 180,E1 -6506.946,E2 -6506.946} C_VEL
LIN {X 0,Y 488.707,Z 259.238,A -85,B 0,C 180,E1 -6510.364,E2 -6510.364} C_VEL
LIN {X 0,Y 488.732,Z 259.237,A -85,B 0,C 180,E1 -6513.485,E2 -6513.485} C_VEL
LIN {X 0,Y 488.68,Z 259.245,A -85,B 0,C 180,E1 -6516.355,E2 -6516.355} C_VEL
LIN {X 0,Y 488.7,Z 259.24,A -85,B 0,C 180,E1 -6519.255,E2 -6519.255} C_VEL
LIN {X 0,Y 488.706,Z 259.237,A -85,B 0,C 180,E1 -6521.601,E2 -6521.601} C_VEL
LIN {X 0,Y 488.713,Z 259.429,A -85,B 0,C 180,E1 -6523.201,E2 -6523.201} C_VEL
LIN {X 0,Y 489.958,Z 265.753,A -85,B 0,C 180,E1 -6526.488,E2 -6526.488} C_VEL
LIN {X 0,Y 490.338,Z 269.259,A -85,B 0,C 180,E1 -6528.187,E2 -6528.187} C_VEL
LIN {X 0,Y 490.267,Z 275.187,A -85,B 0,C 180,E1 -6530.723,E2 -6530.723} C_VEL
LIN {X 0,Y 489.972,Z 281.791,A -85,B 0,C 180,E1 -6533.442,E2 -6533.442} C_VEL
LIN {X 0,Y 489.637,Z 290.839,A -85,B 0,C 180,E1 -6536.947,E2 -6536.947} C_VEL
LIN {X 0,Y 489.344,Z 299.88,A -85,B 0,C 180,E1 -6540.299,E2 -6540.299} C_VEL
LIN {X 0,Y 489.171,Z 307.539,A -85,B 0,C 180,E1 -6542.97,E2 -6542.97} C_VEL
LIN {X 0,Y 488.953,Z 315.835,A -85,B 0,C 180,E1 -6545.818,E2 -6545.818} C_VEL
LIN {X 0,Y 488.766,Z 323.436,A -85,B 0,C 180,E1 -6548.491,E2 -6548.491} C_VEL
LIN {X 0,Y 488.707,Z 325.4,A -85,B 0,C 180,E1 -6549.189,E2 -6549.189} C_VEL
LIN {X 0,Y 493.226,Z 343.451,A -85,B 0,C 180,E1 -6549.759,E2 -6549.759} C_VEL
LIN {X 0,Y 493.888,Z 347.827,A -85,B 0,C 180,E1 -6549.914,E2 -6549.914} C_VEL
LIN {X 0,Y 493.431,Z 362.608,A -85,B 0,C 180,E1 -6550.42,E2 -6550.42} C_VEL
LIN {X 0,Y 492.809,Z 376.823,A -85,B 0,C 180,E1 -6551.069,E2 -6551.069} C_VEL
LIN {X 0,Y 492.097,Z 391.103,A -85,B 0,C 180,E1 -6551.904,E2 -6551.904} C_VEL
LIN {X 0,Y 491.415,Z 404.098,A -85,B 0,C 180,E1 -6552.845,E2 -6552.845} C_VEL
LIN {X 0,Y 490.764,Z 416.648,A -85,B 0,C 180,E1 -6553.948,E2 -6553.948} C_VEL
LIN {X 0,Y 490.097,Z 427.189,A -85,B 0,C 180,E1 -6555.042,E2 -6555.042} C_VEL
LIN {X 0,Y 489.547,Z 437.396,A -85,B 0,C 180,E1 -6556.298,E2 -6556.298} C_VEL
LIN {X 0,Y 488.904,Z 447.766,A -85,B 0,C 180,E1 -6557.823,E2 -6557.823} C_VEL
LIN {X 0,Y 488.705,Z 455.652,A -85,B 0,C 180,E1 -6559.226,E2 -6559.226} C_VEL
LIN {X 0,Y 488.304,Z 463.426,A -85,B 0,C 180,E1 -6560.891,E2 -6560.891} C_VEL
LIN {X 0,Y 488.097,Z 469.608,A -85,B 0,C 180,E1 -6562.555,E2 -6562.555} C_VEL
LIN {X 0,Y 488.033,Z 474.388,A -85,B 0,C 180,E1 -6564.215,E2 -6564.215} C_VEL
LIN {X 0,Y 487.893,Z 477.889,A -85,B 0,C 180,E1 -6565.87,E2 -6565.87} C_VEL
LIN {X 0,Y 487.883,Z 480.19,A -85,B 0,C 180,E1 -6567.524,E2 -6567.524} C_VEL
LIN {X 0,Y 487.831,Z 481.348,A -85,B 0,C 180,E1 -6569.175,E2 -6569.175} C_VEL
LIN {X 0,Y 487.831,Z 481.347,A -85,B 0,C 180,E1 -6570.826,E2 -6570.826} C_VEL
LIN {X 0,Y 487.884,Z 480.186,A -85,B 0,C 180,E1 -6572.477,E2 -6572.477} C_VEL
LIN {X 0,Y 487.893,Z 477.883,A -85,B 0,C 180,E1 -6574.131,E2 -6574.131} C_VEL
LIN {X 0,Y 488.025,Z 474.385,A -85,B 0,C 180,E1 -6575.786,E2 -6575.786} C_VEL
LIN {X 0,Y 488.098,Z 469.607,A -85,B 0,C 180,E1 -6577.446,E2 -6577.446} C_VEL
LIN {X 0,Y 488.305,Z 463.418,A -85,B 0,C 180,E1 -6579.11,E2 -6579.11} C_VEL
LIN {X 0,Y 488.704,Z 455.641,A -85,B 0,C 180,E1 -6580.775,E2 -6580.775} C_VEL
LIN {X 0,Y 488.973,Z 447.53,A -85,B 0,C 180,E1 -6582.214,E2 -6582.214} C_VEL
LIN {X 0,Y 489.547,Z 437.387,A -85,B 0,C 180,E1 -6583.703,E2 -6583.703} C_VEL
LIN {X 0,Y 490.089,Z 427.18,A -85,B 0,C 180,E1 -6584.959,E2 -6584.959} C_VEL
LIN {X 0,Y 490.831,Z 414.805,A -85,B 0,C 180,E1 -6586.234,E2 -6586.234} C_VEL
LIN {X 0,Y 491.554,Z 401.46,A -85,B 0,C 180,E1 -6587.366,E2 -6587.366} C_VEL
LIN {X 0,Y 492.258,Z 387.869,A -85,B 0,C 180,E1 -6588.307,E2 -6588.307} C_VEL
LIN {X 0,Y 492.979,Z 373.789,A -85,B 0,C 180,E1 -6589.087,E2 -6589.087} C_VEL
LIN {X 0,Y 493.516,Z 358.536,A -85,B 0,C 180,E1 -6589.743,E2 -6589.743} C_VEL
LIN {X 0,Y 493.755,Z 345.921,A -85,B 0,C 180,E1 -6590.148,E2 -6590.148} C_VEL
LIN {X 0,Y 490.104,Z 330.965,A -85,B 0,C 180,E1 -6590.647,E2 -6590.647} C_VEL
LIN {X 0,Y 488.694,Z 325.413,A -85,B 0,C 180,E1 -6590.807,E2 -6590.807} C_VEL
LIN {X 0,Y 488.92,Z 317.166,A -85,B 0,C 180,E1 -6593.734,E2 -6593.734} C_VEL
LIN {X 0,Y 489.134,Z 309.354,A -85,B 0,C 180,E1 -6596.45,E2 -6596.45} C_VEL
LIN {X 0,Y 489.401,Z 300.177,A -85,B 0,C 180,E1 -6599.699,E2 -6599.699} C_VEL
LIN {X 0,Y 489.614,Z 292.483,A -85,B 0,C 180,E1 -6602.567,E2 -6602.567} C_VEL
LIN {X 0,Y 489.912,Z 284.904,A -85,B 0,C 180,E1 -6605.538,E2 -6605.538} C_VEL
LIN {X 0,Y 490.307,Z 277.426,A -85,B 0,C 180,E1 -6608.574,E2 -6608.574} C_VEL
LIN {X 0,Y 490.493,Z 271.18,A -85,B 0,C 180,E1 -6611.232,E2 -6611.232} C_VEL
LIN {X 0,Y 490.167,Z 267.278,A -85,B 0,C 180,E1 -6613.009,E2 -6613.009} C_VEL
LIN {X 0,Y 489.114,Z 261.311,A -85,B 0,C 180,E1 -6615.927,E2 -6615.927} C_VEL
LIN {X 0,Y 488.694,Z 259.239,A -85,B 0,C 180,E1 -6617.021,E2 -6617.021} C_VEL
LIN {X 0,Y 488.738,Z 259.234,A -85,B 0,C 180,E1 -6619.677,E2 -6619.677} C_VEL
LIN {X 0,Y 488.684,Z 259.239,A -85,B 0,C 180,E1 -6622.841,E2 -6622.841} C_VEL
LIN {X 0,Y 488.729,Z 259.234,A -85,B 0,C 180,E1 -6625.887,E2 -6625.887} C_VEL
LIN {X 0,Y 488.698,Z 259.24,A -85,B 0,C 180,E1 -6628.82,E2 -6628.82} C_VEL
LIN {X 0,Y 488.748,Z 259.23,A -85,B 0,C 180,E1 -6631.671,E2 -6631.671} C_VEL
LIN {X 0,Y 488.753,Z 259.231,A -85,B 0,C 180,E1 -6634.444,E2 -6634.444} C_VEL
LIN {X 0,Y 488.728,Z 259.234,A -85,B 0,C 180,E1 -6637.153,E2 -6637.153} C_VEL
LIN {X 0,Y 488.731,Z 259.231,A -85,B 0,C 180,E1 -6639.81,E2 -6639.81} C_VEL
LIN {X 0,Y 488.74,Z 259.234,A -85,B 0,C 180,E1 -6642.423,E2 -6642.423} C_VEL
LIN {X 0,Y 488.767,Z 259.229,A -85,B 0,C 180,E1 -6644.999,E2 -6644.999} C_VEL
LIN {X 0,Y 488.811,Z 259.224,A -85,B 0,C 180,E1 -6648.387,E2 -6648.387} C_VEL
LIN {X 0,Y 488.821,Z 259.221,A -85,B 0,C 180,E1 -6651.733,E2 -6651.733} C_VEL
LIN {X 0,Y 488.811,Z 259.222,A -85,B 0,C 180,E1 -6655.05,E2 -6655.05} C_VEL
LIN {X 0,Y 488.965,Z 259.202,A -85,B 0,C 180,E1 -6657.528,E2 -6657.528} C_VEL
LIN {X 0,Y 488.959,Z 259.205,A -85,B 0,C 180,E1 -6660.823,E2 -6660.823} C_VEL
LIN {X 0,Y 488.963,Z 259.205,A -85,B 0,C 180,E1 -6662.47,E2 -6662.47} C_VEL
LIN {X 0,Y 488.857,Z 259.218,A -85,B 0,C 180,E1 -6665.775,E2 -6665.775} C_VEL
LIN {X 0,Y 488.82,Z 259.223,A -85,B 0,C 180,E1 -6668.265,E2 -6668.265} C_VEL
LIN {X 0,Y 488.808,Z 259.223,A -85,B 0,C 180,E1 -6671.611,E2 -6671.611} C_VEL
LIN {X 0,Y 488.764,Z 259.228,A -85,B 0,C 180,E1 -6674.999,E2 -6674.999} C_VEL
LIN {X 0,Y 488.756,Z 259.23,A -85,B 0,C 180,E1 -6678.441,E2 -6678.441} C_VEL
LIN {X 0,Y 488.707,Z 259.235,A -85,B 0,C 180,E1 -6681.069,E2 -6681.069} C_VEL
LIN {X 0,Y 488.693,Z 259.238,A -85,B 0,C 180,E1 -6683.744,E2 -6683.744} C_VEL
LIN {X 0,Y 488.791,Z 259.224,A -85,B 0,C 180,E1 -6686.942,E2 -6686.942} C_VEL
LIN {X 0,Y 488.708,Z 259.238,A -85,B 0,C 180,E1 -6690.362,E2 -6690.362} C_VEL
LIN {X 0,Y 488.734,Z 259.232,A -85,B 0,C 180,E1 -6693.483,E2 -6693.483} C_VEL
LIN {X 0,Y 488.686,Z 259.239,A -85,B 0,C 180,E1 -6696.354,E2 -6696.354} C_VEL
LIN {X 0,Y 488.698,Z 259.237,A -85,B 0,C 180,E1 -6699.253,E2 -6699.253} C_VEL
LIN {X 0,Y 488.719,Z 259.235,A -85,B 0,C 180,E1 -6701.601,E2 -6701.601} C_VEL
LIN {X 0,Y 488.707,Z 259.235,A -85,B 0,C 180,E1 -6704.8,E2 -6704.8} C_VEL
LIN {X 0,Y 488.726,Z 259.235,A -85,B 0,C 180,E1 -6707.478,E2 -6707.478} C_VEL
LIN {X 0,Y 488.736,Z 259.231,A -85,B 0,C 180,E1 -6710.749,E2 -6710.749} C_VEL
LIN {X 0,Y 488.679,Z 259.24,A -85,B 0,C 180,E1 -6713.868,E2 -6713.868} C_VEL
LIN {X 0,Y 488.732,Z 259.232,A -85,B 0,C 180,E1 -6716.876,E2 -6716.876} C_VEL
LIN {X 0,Y 488.726,Z 259.236,A -85,B 0,C 180,E1 -6719.78,E2 -6719.78} C_VEL
LIN {X 0,Y 488.791,Z 259.226,A -85,B 0,C 180,E1 -6723.054,E2 -6723.054} C_VEL
LIN {X 0,Y 488.738,Z 259.23,A -85,B 0,C 180,E1 -6724.343,E2 -6724.343} C_VEL
LIN {X 0,Y 488.09,Z 259.314,A -85,B 0,C 180,E1 -6725.031,E2 -6725.031} C_VEL
LIN {X 0,Y 485.22,Z 259.674,A -85,B 0,C 180,E1 -6726.147,E2 -6726.147} C_VEL
LIN {X 0,Y 482.774,Z 259.978,A -85,B 0,C 180,E1 -6727.047,E2 -6727.047} C_VEL
LIN {X 0,Y 481.717,Z 260.108,A -85,B 0,C 180,E1 -6727.742,E2 -6727.742} C_VEL
LIN {X 0,Y 481.628,Z 260.116,A -85,B 0,C 180,E1 -6727.978,E2 -6727.978} C_VEL
LIN {X 0,Y 481.699,Z 260.108,A -85,B 0,C 180,E1 -6730.392,E2 -6730.392} C_VEL
LIN {X 0,Y 481.682,Z 260.111,A -85,B 0,C 180,E1 -6733.033,E2 -6733.033} C_VEL
LIN {X 0,Y 481.684,Z 260.112,A -85,B 0,C 180,E1 -6735.638,E2 -6735.638} C_VEL
LIN {X 0,Y 481.785,Z 260.097,A -85,B 0,C 180,E1 -6738.215,E2 -6738.215} C_VEL
LIN {X 0,Y 481.754,Z 260.104,A -85,B 0,C 180,E1 -6741.611,E2 -6741.611} C_VEL
LIN {X 0,Y 481.791,Z 260.095,A -85,B 0,C 180,E1 -6744.139,E2 -6744.139} C_VEL
LIN {X 0,Y 481.408,Z 260.147,A -85,B 0,C 180,E1 -6746.652,E2 -6746.652} C_VEL
LIN {X 0,Y 481.462,Z 260.242,A -85,B 0,C 180,E1 -6748.326,E2 -6748.326} C_VEL
LIN {X 0,Y 481.56,Z 261.757,A -85,B 0,C 180,E1 -6749.999,E2 -6749.999} C_VEL
LIN {X 0,Y 481.317,Z 265.689,A -85,B 0,C 180,E1 -6754.186,E2 -6754.186} C_VEL
LIN {X 0,Y 481.163,Z 268.863,A -85,B 0,C 180,E1 -6757.553,E2 -6757.553} C_VEL
LIN {X 0,Y 481.117,Z 272.079,A -85,B 0,C 180,E1 -6760.946,E2 -6760.946} C_VEL
LIN {X 0,Y 481.116,Z 273.109,A -85,B 0,C 180,E1 -6761.987,E2 -6761.987} C_VEL
LIN {X 0,Y 485.886,Z 288.439,A -85,B 0,C 180,E1 -6762.55,E2 -6762.55} C_VEL
LIN {X 0,Y 487.213,Z 293.921,A -85,B 0,C 180,E1 -6762.777,E2 -6762.777} C_VEL
LIN {X 0,Y 486.718,Z 307.606,A -85,B 0,C 180,E1 -6763.278,E2 -6763.278} C_VEL
LIN {X 0,Y 486.181,Z 321.115,A -85,B 0,C 180,E1 -6763.926,E2 -6763.926} C_VEL
LIN {X 0,Y 485.504,Z 334.774,A -85,B 0,C 180,E1 -6764.749,E2 -6764.749} C_VEL
LIN {X 0,Y 484.797,Z 348.449,A -85,B 0,C 180,E1 -6765.772,E2 -6765.772} C_VEL
LIN {X 0,Y 484.109,Z 360.62,A -85,B 0,C 180,E1 -6766.878,E2 -6766.878} C_VEL
LIN {X 0,Y 483.301,Z 372.864,A -85,B 0,C 180,E1 -6768.218,E2 -6768.218} C_VEL
LIN {X 0,Y 482.673,Z 383.093,A -85,B 0,C 180,E1 -6769.565,E2 -6769.565} C_VEL
LIN {X 0,Y 482.096,Z 392.785,A -85,B 0,C 180,E1 -6771.098,E2 -6771.098} C_VEL
LIN {X 0,Y 481.671,Z 401.248,A -85,B 0,C 180,E1 -6772.728,E2 -6772.728} C_VEL
LIN {X 0,Y 481.378,Z 407.264,A -85,B 0,C 180,E1 -6774.128,E2 -6774.128} C_VEL
LIN {X 0,Y 481.175,Z 412.21,A -85,B 0,C 180,E1 -6775.522,E2 -6775.522} C_VEL
LIN {X 0,Y 481.039,Z 416.337,A -85,B 0,C 180,E1 -6776.977,E2 -6776.977} C_VEL
LIN {X 0,Y 480.83,Z 420.264,A -85,B 0,C 180,E1 -6778.838,E2 -6778.838} C_VEL
LIN {X 0,Y 480.755,Z 422.803,A -85,B 0,C 180,E1 -6780.773,E2 -6780.773} C_VEL
LIN {X 0,Y 480.747,Z 423.665,A -85,B 0,C 180,E1 -6782.019,E2 -6782.019} C_VEL
LIN {X 0,Y 480.754,Z 423.773,A -85,B 0,C 180,E1 -6783.745,E2 -6783.745} C_VEL
LIN {X 0,Y 480.758,Z 423.093,A -85,B 0,C 180,E1 -6785.054,E2 -6785.054} C_VEL
LIN {X 0,Y 480.789,Z 421.082,A -85,B 0,C 180,E1 -6786.821,E2 -6786.821} C_VEL
LIN {X 0,Y 481.002,Z 418.163,A -85,B 0,C 180,E1 -6788.386,E2 -6788.386} C_VEL
LIN {X 0,Y 481.096,Z 414.072,A -85,B 0,C 180,E1 -6789.997,E2 -6789.997} C_VEL
LIN {X 0,Y 481.315,Z 409.261,A -85,B 0,C 180,E1 -6791.478,E2 -6791.478} C_VEL
LIN {X 0,Y 481.623,Z 402.479,A -85,B 0,C 180,E1 -6793.148,E2 -6793.148} C_VEL
LIN {X 0,Y 482.081,Z 394.706,A -85,B 0,C 180,E1 -6794.7,E2 -6794.7} C_VEL
LIN {X 0,Y 482.596,Z 386.133,A -85,B 0,C 180,E1 -6796.124,E2 -6796.124} C_VEL
LIN {X 0,Y 483.202,Z 375.572,A -85,B 0,C 180,E1 -6797.586,E2 -6797.586} C_VEL
LIN {X 0,Y 483.915,Z 364.562,A -85,B 0,C 180,E1 -6798.853,E2 -6798.853} C_VEL
LIN {X 0,Y 484.679,Z 352.386,A -85,B 0,C 180,E1 -6800.022,E2 -6800.022} C_VEL
LIN {X 0,Y 485.419,Z 339.06,A -85,B 0,C 180,E1 -6801.079,E2 -6801.079} C_VEL
LIN {X 0,Y 486.128,Z 325.318,A -85,B 0,C 180,E1 -6801.96,E2 -6801.96} C_VEL
LIN {X 0,Y 486.709,Z 311.451,A -85,B 0,C 180,E1 -6802.667,E2 -6802.667} C_VEL
LIN {X 0,Y 487.218,Z 295.973,A -85,B 0,C 180,E1 -6803.266,E2 -6803.266} C_VEL
LIN {X 0,Y 486.999,Z 292.335,A -85,B 0,C 180,E1 -6803.388,E2 -6803.388} C_VEL
LIN {X 0,Y 482.529,Z 278.46,A -85,B 0,C 180,E1 -6803.95,E2 -6803.95} C_VEL
LIN {X 0,Y 481.102,Z 273.918,A -85,B 0,C 180,E1 -6804.117,E2 -6804.117} C_VEL
LIN {X 0,Y 481.184,Z 271.056,A -85,B 0,C 180,E1 -6807.29,E2 -6807.29} C_VEL
LIN {X 0,Y 481.237,Z 268.432,A -85,B 0,C 180,E1 -6810.23,E2 -6810.23} C_VEL
LIN {X 0,Y 481.299,Z 265.917,A -85,B 0,C 180,E1 -6813.087,E2 -6813.087} C_VEL
LIN {X 0,Y 481.368,Z 263.434,A -85,B 0,C 180,E1 -6815.872,E2 -6815.872} C_VEL
LIN {X 0,Y 481.427,Z 260.574,A -85,B 0,C 180,E1 -6819.112,E2 -6819.112} C_VEL
LIN {X 0,Y 481.453,Z 260.237,A -85,B 0,C 180,E1 -6819.493,E2 -6819.493} C_VEL
LIN {X 0,Y 481.641,Z 260.12,A -85,B 0,C 180,E1 -6822.157,E2 -6822.157} C_VEL
LIN {X 0,Y 481.735,Z 260.107,A -85,B 0,C 180,E1 -6824.777,E2 -6824.777} C_VEL
LIN {X 0,Y 481.744,Z 260.104,A -85,B 0,C 180,E1 -6828.216,E2 -6828.216} C_VEL
LIN {X 0,Y 481.758,Z 260.102,A -85,B 0,C 180,E1 -6831.613,E2 -6831.613} C_VEL
LIN {X 0,Y 481.812,Z 260.096,A -85,B 0,C 180,E1 -6834.141,E2 -6834.141} C_VEL
LIN {X 0,Y 481.925,Z 260.081,A -85,B 0,C 180,E1 -6837.493,E2 -6837.493} C_VEL
LIN {X 0,Y 481.902,Z 260.084,A -85,B 0,C 180,E1 -6840.837,E2 -6840.837} C_VEL
LIN {X 0,Y 481.924,Z 260.082,A -85,B 0,C 180,E1 -6842.508,E2 -6842.508} C_VEL
LIN {X 0,Y 481.814,Z 260.094,A -85,B 0,C 180,E1 -6845.861,E2 -6845.861} C_VEL
LIN {X 0,Y 481.76,Z 260.1,A -85,B 0,C 180,E1 -6848.389,E2 -6848.389} C_VEL
LIN {X 0,Y 481.748,Z 260.103,A -85,B 0,C 180,E1 -6851.786,E2 -6851.786} C_VEL
LIN {X 0,Y 481.739,Z 260.103,A -85,B 0,C 180,E1 -6855.225,E2 -6855.225} C_VEL
LIN {X 0,Y 481.709,Z 260.107,A -85,B 0,C 180,E1 -6858.722,E2 -6858.722} C_VEL
LIN {X 0,Y 481.645,Z 260.116,A -85,B 0,C 180,E1 -6861.395,E2 -6861.395} C_VEL
LIN {X 0,Y 481.675,Z 260.112,A -85,B 0,C 180,E1 -6864.114,E2 -6864.114} C_VEL
LIN {X 0,Y 481.75,Z 260.102,A -85,B 0,C 180,E1 -6867.141,E2 -6867.141} C_VEL
LIN {X 0,Y 481.676,Z 260.115,A -85,B 0,C 180,E1 -6869.742,E2 -6869.742} C_VEL
LIN {X 0,Y 481.669,Z 260.117,A -85,B 0,C 180,E1 -6872.675,E2 -6872.675} C_VEL
LIN {X 0,Y 481.634,Z 260.123,A -85,B 0,C 180,E1 -6875.71,E2 -6875.71} C_VEL
LIN {X 0,Y 481.67,Z 260.117,A -85,B 0,C 180,E1 -6878.86,E2 -6878.86} C_VEL
LIN {X 0,Y 481.651,Z 260.117,A -85,B 0,C 180,E1 -6881.914,E2 -6881.914} C_VEL
LIN {X 0,Y 481.702,Z 260.262,A -85,B 0,C 180,E1 -6882.792,E2 -6882.792} C_VEL
LIN {X 0,Y 482.712,Z 265.652,A -85,B 0,C 180,E1 -6885.666,E2 -6885.666} C_VEL
LIN {X 0,Y 483.38,Z 270.346,A -85,B 0,C 180,E1 -6888.026,E2 -6888.026} C_VEL
LIN {X 0,Y 483.319,Z 275.749,A -85,B 0,C 180,E1 -6890.415,E2 -6890.415} C_VEL
LIN {X 0,Y 482.969,Z 282.831,A -85,B 0,C 180,E1 -6893.373,E2 -6893.373} C_VEL
LIN {X 0,Y 482.63,Z 291.805,A -85,B 0,C 180,E1 -6896.903,E2 -6896.903} C_VEL
LIN {X 0,Y 482.31,Z 300.798,A -85,B 0,C 180,E1 -6900.302,E2 -6900.302} C_VEL
LIN {X 0,Y 482.094,Z 308.807,A -85,B 0,C 180,E1 -6903.134,E2 -6903.134} C_VEL
LIN {X 0,Y 481.854,Z 318.068,A -85,B 0,C 180,E1 -6906.354,E2 -6906.354} C_VEL
LIN {X 0,Y 481.681,Z 325.41,A -85,B 0,C 180,E1 -6908.878,E2 -6908.878} C_VEL
LIN {X 0,Y 485.904,Z 341.945,A -85,B 0,C 180,E1 -6909.403,E2 -6909.403} C_VEL
LIN {X 0,Y 487.221,Z 348.152,A -85,B 0,C 180,E1 -6909.637,E2 -6909.637} C_VEL
LIN {X 0,Y 486.742,Z 361.819,A -85,B 0,C 180,E1 -6910.107,E2 -6910.107} C_VEL
LIN {X 0,Y 486.079,Z 376.822,A -85,B 0,C 180,E1 -6910.797,E2 -6910.797} C_VEL
LIN {X 0,Y 485.339,Z 391.102,A -85,B 0,C 180,E1 -6911.643,E2 -6911.643} C_VEL
LIN {X 0,Y 484.593,Z 404.096,A -85,B 0,C 180,E1 -6912.596,E2 -6912.596} C_VEL
LIN {X 0,Y 483.872,Z 417.009,A -85,B 0,C 180,E1 -6913.749,E2 -6913.749} C_VEL
LIN {X 0,Y 483.073,Z 428.971,A -85,B 0,C 180,E1 -6915.035,E2 -6915.035} C_VEL
LIN {X 0,Y 482.496,Z 438.908,A -85,B 0,C 180,E1 -6916.309,E2 -6916.309} C_VEL
LIN {X 0,Y 481.876,Z 448.299,A -85,B 0,C 180,E1 -6917.735,E2 -6917.735} C_VEL
LIN {X 0,Y 481.621,Z 456.728,A -85,B 0,C 180,E1 -6919.278,E2 -6919.278} C_VEL
LIN {X 0,Y 481.247,Z 463.426,A -85,B 0,C 180,E1 -6920.757,E2 -6920.757} C_VEL
LIN {X 0,Y 481.015,Z 469.608,A -85,B 0,C 180,E1 -6922.445,E2 -6922.445} C_VEL
LIN {X 0,Y 480.941,Z 474.388,A -85,B 0,C 180,E1 -6924.129,E2 -6924.129} C_VEL
LIN {X 0,Y 480.797,Z 477.888,A -85,B 0,C 180,E1 -6925.809,E2 -6925.809} C_VEL
LIN {X 0,Y 480.8,Z 480.19,A -85,B 0,C 180,E1 -6927.487,E2 -6927.487} C_VEL
LIN {X 0,Y 480.757,Z 481.348,A -85,B 0,C 180,E1 -6929.163,E2 -6929.163} C_VEL
LIN {X 0,Y 480.757,Z 481.347,A -85,B 0,C 180,E1 -6930.838,E2 -6930.838} C_VEL
LIN {X 0,Y 480.8,Z 480.186,A -85,B 0,C 180,E1 -6932.514,E2 -6932.514} C_VEL
LIN {X 0,Y 480.797,Z 477.882,A -85,B 0,C 180,E1 -6934.192,E2 -6934.192} C_VEL
LIN {X 0,Y 480.926,Z 474.385,A -85,B 0,C 180,E1 -6935.872,E2 -6935.872} C_VEL
LIN {X 0,Y 481.016,Z 469.607,A -85,B 0,C 180,E1 -6937.557,E2 -6937.557} C_VEL
LIN {X 0,Y 481.248,Z 463.418,A -85,B 0,C 180,E1 -6939.245,E2 -6939.245} C_VEL
LIN {X 0,Y 481.65,Z 455.64,A -85,B 0,C 180,E1 -6940.935,E2 -6940.935} C_VEL
LIN {X 0,Y 482.013,Z 447.058,A -85,B 0,C 180,E1 -6942.468,E2 -6942.468} C_VEL
LIN {X 0,Y 482.615,Z 437.387,A -85,B 0,C 180,E1 -6943.904,E2 -6943.904} C_VEL
LIN {X 0,Y 483.172,Z 427.18,A -85,B 0,C 180,E1 -6945.179,E2 -6945.179} C_VEL
LIN {X 0,Y 483.916,Z 415.547,A -85,B 0,C 180,E1 -6946.398,E2 -6946.398} C_VEL
LIN {X 0,Y 484.662,Z 402.797,A -85,B 0,C 180,E1 -6947.512,E2 -6947.512} C_VEL
LIN {X 0,Y 485.413,Z 389.497,A -85,B 0,C 180,E1 -6948.465,E2 -6948.465} C_VEL
LIN {X 0,Y 486.06,Z 376.797,A -85,B 0,C 180,E1 -6949.205,E2 -6949.205} C_VEL
LIN {X 0,Y 486.696,Z 362.809,A -85,B 0,C 180,E1 -6949.854,E2 -6949.854} C_VEL
LIN {X 0,Y 487.143,Z 347.46,A -85,B 0,C 180,E1 -6950.388,E2 -6950.388} C_VEL
LIN {X 0,Y 483.4,Z 332.035,A -85,B 0,C 180,E1 -6950.926,E2 -6950.926} C_VEL
LIN {X 0,Y 481.68,Z 325.357,A -85,B 0,C 180,E1 -6951.141,E2 -6951.141} C_VEL
LIN {X 0,Y 481.9,Z 316.859,A -85,B 0,C 180,E1 -6954.102,E2 -6954.102} C_VEL
LIN {X 0,Y 482.126,Z 309.04,A -85,B 0,C 180,E1 -6956.866,E2 -6956.866} C_VEL
LIN {X 0,Y 482.36,Z 301.171,A -85,B 0,C 180,E1 -6959.695,E2 -6959.695} C_VEL
LIN {X 0,Y 482.598,Z 293.509,A -85,B 0,C 180,E1 -6962.604,E2 -6962.604} C_VEL
LIN {X 0,Y 482.92,Z 285.974,A -85,B 0,C 180,E1 -6965.601,E2 -6965.601} C_VEL
LIN {X 0,Y 483.353,Z 278.456,A -85,B 0,C 180,E1 -6968.699,E2 -6968.699} C_VEL
LIN {X 0,Y 483.525,Z 272.231,A -85,B 0,C 180,E1 -6971.402,E2 -6971.402} C_VEL
LIN {X 0,Y 483.14,Z 268.066,A -85,B 0,C 180,E1 -6973.337,E2 -6973.337} C_VEL
LIN {X 0,Y 482.107,Z 262.383,A -85,B 0,C 180,E1 -6976.176,E2 -6976.176} C_VEL
LIN {X 0,Y 481.651,Z 260.117,A -85,B 0,C 180,E1 -6977.454,E2 -6977.454} C_VEL
LIN {X 0,Y 481.685,Z 260.113,A -85,B 0,C 180,E1 -6980.651,E2 -6980.651} C_VEL
LIN {X 0,Y 481.633,Z 260.118,A -85,B 0,C 180,E1 -6983.376,E2 -6983.376} C_VEL
LIN {X 0,Y 481.682,Z 260.111,A -85,B 0,C 180,E1 -6986.327,E2 -6986.327} C_VEL
LIN {X 0,Y 481.656,Z 260.114,A -85,B 0,C 180,E1 -6989.417,E2 -6989.417} C_VEL
LIN {X 0,Y 481.704,Z 260.108,A -85,B 0,C 180,E1 -6992.168,E2 -6992.168} C_VEL
LIN {X 0,Y 481.723,Z 260.108,A -85,B 0,C 180,E1 -6994.97,E2 -6994.97} C_VEL
LIN {X 0,Y 481.655,Z 260.112,A -85,B 0,C 180,E1 -6997.704,E2 -6997.704} C_VEL
LIN {X 0,Y 481.712,Z 260.109,A -85,B 0,C 180,E1 -7000.393,E2 -7000.393} C_VEL
LIN {X 0,Y 481.697,Z 260.11,A -85,B 0,C 180,E1 -7003.033,E2 -7003.033} C_VEL
LIN {X 0,Y 481.694,Z 260.109,A -85,B 0,C 180,E1 -7005.638,E2 -7005.638} C_VEL
LIN {X 0,Y 481.756,Z 260.102,A -85,B 0,C 180,E1 -7008.214,E2 -7008.214} C_VEL
LIN {X 0,Y 481.767,Z 260.099,A -85,B 0,C 180,E1 -7011.611,E2 -7011.611} C_VEL
LIN {X 0,Y 481.781,Z 260.099,A -85,B 0,C 180,E1 -7014.978,E2 -7014.978} C_VEL
LIN {X 0,Y 481.932,Z 260.078,A -85,B 0,C 180,E1 -7017.492,E2 -7017.492} C_VEL
LIN {X 0,Y 481.91,Z 260.083,A -85,B 0,C 180,E1 -7020.835,E2 -7020.835} C_VEL
LIN {X 0,Y 481.93,Z 260.081,A -85,B 0,C 180,E1 -7022.507,E2 -7022.507} C_VEL
LIN {X 0,Y 481.819,Z 260.095,A -85,B 0,C 180,E1 -7025.859,E2 -7025.859} C_VEL
LIN {X 0,Y 481.766,Z 260.103,A -85,B 0,C 180,E1 -7028.387,E2 -7028.387} C_VEL
LIN {X 0,Y 481.753,Z 260.103,A -85,B 0,C 180,E1 -7031.784,E2 -7031.784} C_VEL
LIN {X 0,Y 481.745,Z 260.101,A -85,B 0,C 180,E1 -7035.223,E2 -7035.223} C_VEL
LIN {X 0,Y 481.713,Z 260.108,A -85,B 0,C 180,E1 -7038.72,E2 -7038.72} C_VEL
LIN {X 0,Y 481.646,Z 260.115,A -85,B 0,C 180,E1 -7041.393,E2 -7041.393} C_VEL
LIN {X 0,Y 481.677,Z 260.114,A -85,B 0,C 180,E1 -7044.112,E2 -7044.112} C_VEL
LIN {X 0,Y 481.746,Z 260.102,A -85,B 0,C 180,E1 -7047.138,E2 -7047.138} C_VEL
LIN {X 0,Y 481.677,Z 260.113,A -85,B 0,C 180,E1 -7049.74,E2 -7049.74} C_VEL
LIN {X 0,Y 481.67,Z 260.112,A -85,B 0,C 180,E1 -7052.673,E2 -7052.673} C_VEL
LIN {X 0,Y 481.64,Z 260.118,A -85,B 0,C 180,E1 -7055.708,E2 -7055.708} C_VEL
LIN {X 0,Y 481.668,Z 260.112,A -85,B 0,C 180,E1 -7058.858,E2 -7058.858} C_VEL
LIN {X 0,Y 481.658,Z 260.116,A -85,B 0,C 180,E1 -7061.913,E2 -7061.913} C_VEL
LIN {X 0,Y 481.655,Z 260.113,A -85,B 0,C 180,E1 -7064.456,E2 -7064.456} C_VEL
LIN {X 0,Y 481.683,Z 260.109,A -85,B 0,C 180,E1 -7066.844,E2 -7066.844} C_VEL
LIN {X 0,Y 481.683,Z 260.112,A -85,B 0,C 180,E1 -7070.06,E2 -7070.06} C_VEL
LIN {X 0,Y 481.623,Z 260.118,A -85,B 0,C 180,E1 -7073.252,E2 -7073.252} C_VEL
LIN {X 0,Y 481.702,Z 260.109,A -85,B 0,C 180,E1 -7076.329,E2 -7076.329} C_VEL
LIN {X 0,Y 481.651,Z 260.116,A -85,B 0,C 180,E1 -7079.414,E2 -7079.414} C_VEL
LIN {X 0,Y 481.695,Z 260.109,A -85,B 0,C 180,E1 -7082.167,E2 -7082.167} C_VEL
LIN {X 0,Y 481.71,Z 260.107,A -85,B 0,C 180,E1 -7084.969,E2 -7084.969} C_VEL
LIN {X 0,Y 481.628,Z 260.116,A -85,B 0,C 180,E1 -7087.978,E2 -7087.978} C_VEL
LIN {X 0,Y 480.96,Z 260.199,A -85,B 0,C 180,E1 -7088.676,E2 -7088.676} C_VEL
LIN {X 0,Y 478.133,Z 260.554,A -85,B 0,C 180,E1 -7089.81,E2 -7089.81} C_VEL
LIN {X 0,Y 475.748,Z 260.852,A -85,B 0,C 180,E1 -7090.724,E2 -7090.724} C_VEL
LIN {X 0,Y 474.727,Z 260.979,A -85,B 0,C 180,E1 -7091.43,E2 -7091.43} C_VEL
LIN {X 0,Y 474.646,Z 260.988,A -85,B 0,C 180,E1 -7091.669,E2 -7091.669} C_VEL
LIN {X 0,Y 474.69,Z 260.981,A -85,B 0,C 180,E1 -7094.543,E2 -7094.543} C_VEL
LIN {X 0,Y 474.729,Z 260.977,A -85,B 0,C 180,E1 -7098.038,E2 -7098.038} C_VEL
LIN {X 0,Y 474.719,Z 260.98,A -85,B 0,C 180,E1 -7101.486,E2 -7101.486} C_VEL
LIN {X 0,Y 474.756,Z 260.972,A -85,B 0,C 180,E1 -7104.052,E2 -7104.052} C_VEL
LIN {X 0,Y 474.367,Z 261.023,A -85,B 0,C 180,E1 -7106.602,E2 -7106.602} C_VEL
LIN {X 0,Y 474.4,Z 261.021,A -85,B 0,C 180,E1 -7108.302,E2 -7108.302} C_VEL
LIN {X 0,Y 474.606,Z 261.749,A -85,B 0,C 180,E1 -7109.151,E2 -7109.151} C_VEL
LIN {X 0,Y 474.404,Z 263.324,A -85,B 0,C 180,E1 -7110.848,E2 -7110.848} C_VEL
LIN {X 0,Y 474.256,Z 266.477,A -85,B 0,C 180,E1 -7114.249,E2 -7114.249} C_VEL
LIN {X 0,Y 474.108,Z 269.689,A -85,B 0,C 180,E1 -7117.666,E2 -7117.666} C_VEL
LIN {X 0,Y 474.097,Z 273.434,A -85,B 0,C 180,E1 -7121.632,E2 -7121.632} C_VEL
LIN {X 0,Y 474.147,Z 273.962,A -85,B 0,C 180,E1 -7121.674,E2 -7121.674} C_VEL
LIN {X 0,Y 479.073,Z 289.34,A -85,B 0,C 180,E1 -7122.264,E2 -7122.264} C_VEL
LIN {X 0,Y 480.559,Z 295.368,A -85,B 0,C 180,E1 -7122.52,E2 -7122.52} C_VEL
LIN {X 0,Y 479.999,Z 310.205,A -85,B 0,C 180,E1 -7123.089,E2 -7123.089} C_VEL
LIN {X 0,Y 479.371,Z 323.434,A -85,B 0,C 180,E1 -7123.756,E2 -7123.756} C_VEL
LIN {X 0,Y 478.611,Z 337.906,A -85,B 0,C 180,E1 -7124.672,E2 -7124.672} C_VEL
LIN {X 0,Y 477.943,Z 350.657,A -85,B 0,C 180,E1 -7125.675,E2 -7125.675} C_VEL
LIN {X 0,Y 477.151,Z 362.491,A -85,B 0,C 180,E1 -7126.791,E2 -7126.791} C_VEL
LIN {X 0,Y 476.395,Z 373.635,A -85,B 0,C 180,E1 -7128.047,E2 -7128.047} C_VEL
LIN {X 0,Y 475.736,Z 383.83,A -85,B 0,C 180,E1 -7129.416,E2 -7129.416} C_VEL
LIN {X 0,Y 475.175,Z 392.453,A -85,B 0,C 180,E1 -7130.791,E2 -7130.791} C_VEL
LIN {X 0,Y 474.71,Z 400.893,A -85,B 0,C 180,E1 -7132.409,E2 -7132.409} C_VEL
LIN {X 0,Y 474.351,Z 407.863,A -85,B 0,C 180,E1 -7134.043,E2 -7134.043} C_VEL
LIN {X 0,Y 474.124,Z 412.795,A -85,B 0,C 180,E1 -7135.459,E2 -7135.459} C_VEL
LIN {X 0,Y 473.953,Z 417.456,A -85,B 0,C 180,E1 -7137.167,E2 -7137.167} C_VEL
LIN {X 0,Y 473.757,Z 420.958,A -85,B 0,C 180,E1 -7138.93,E2 -7138.93} C_VEL
LIN {X 0,Y 473.707,Z 423.137,A -85,B 0,C 180,E1 -7140.631,E2 -7140.631} C_VEL
LIN {X 0,Y 473.649,Z 424.19,A -85,B 0,C 180,E1 -7142.287,E2 -7142.287} C_VEL
LIN {X 0,Y 473.671,Z 424.207,A -85,B 0,C 180,E1 -7143.813,E2 -7143.813} C_VEL
LIN {X 0,Y 473.677,Z 423.292,A -85,B 0,C 180,E1 -7145.355,E2 -7145.355} C_VEL
LIN {X 0,Y 473.704,Z 421.693,A -85,B 0,C 180,E1 -7146.762,E2 -7146.762} C_VEL
LIN {X 0,Y 473.931,Z 418.498,A -85,B 0,C 180,E1 -7148.522,E2 -7148.522} C_VEL
LIN {X 0,Y 474.057,Z 414.362,A -85,B 0,C 180,E1 -7150.157,E2 -7150.157} C_VEL
LIN {X 0,Y 474.304,Z 408.922,A -85,B 0,C 180,E1 -7151.819,E2 -7151.819} C_VEL
LIN {X 0,Y 474.642,Z 402.057,A -85,B 0,C 180,E1 -7153.488,E2 -7153.488} C_VEL
LIN {X 0,Y 475.128,Z 394.852,A -85,B 0,C 180,E1 -7154.927,E2 -7154.927} C_VEL
LIN {X 0,Y 475.722,Z 385.164,A -85,B 0,C 180,E1 -7156.529,E2 -7156.529} C_VEL
LIN {X 0,Y 476.42,Z 374.419,A -85,B 0,C 180,E1 -7157.996,E2 -7157.996} C_VEL
LIN {X 0,Y 477.218,Z 362.663,A -85,B 0,C 180,E1 -7159.326,E2 -7159.326} C_VEL
LIN {X 0,Y 478.072,Z 349.957,A -85,B 0,C 180,E1 -7160.514,E2 -7160.514} C_VEL
LIN {X 0,Y 478.842,Z 336.554,A -85,B 0,C 180,E1 -7161.544,E2 -7161.544} C_VEL
LIN {X 0,Y 479.605,Z 322.347,A -85,B 0,C 180,E1 -7162.42,E2 -7162.42} C_VEL
LIN {X 0,Y 480.179,Z 307.806,A -85,B 0,C 180,E1 -7163.126,E2 -7163.126} C_VEL
LIN {X 0,Y 480.568,Z 294.667,A -85,B 0,C 180,E1 -7163.613,E2 -7163.613} C_VEL
LIN {X 0,Y 475.985,Z 280.25,A -85,B 0,C 180,E1 -7164.226,E2 -7164.226} C_VEL
LIN {X 0,Y 474.049,Z 274.415,A -85,B 0,C 180,E1 -7164.443,E2 -7164.443} C_VEL
LIN {X 0,Y 474.17,Z 271.455,A -85,B 0,C 180,E1 -7167.754,E2 -7167.754} C_VEL
LIN {X 0,Y 474.226,Z 268.596,A -85,B 0,C 180,E1 -7170.97,E2 -7170.97} C_VEL
LIN {X 0,Y 474.252,Z 266.301,A -85,B 0,C 180,E1 -7173.605,E2 -7173.605} C_VEL
LIN {X 0,Y 474.351,Z 263.569,A -85,B 0,C 180,E1 -7176.719,E2 -7176.719} C_VEL
LIN {X 0,Y 474.393,Z 261.413,A -85,B 0,C 180,E1 -7179.174,E2 -7179.174} C_VEL
LIN {X 0,Y 474.537,Z 261.005,A -85,B 0,C 180,E1 -7180.986,E2 -7180.986} C_VEL
LIN {X 0,Y 474.673,Z 260.987,A -85,B 0,C 180,E1 -7184.233,E2 -7184.233} C_VEL
LIN {X 0,Y 474.694,Z 260.984,A -85,B 0,C 180,E1 -7187.725,E2 -7187.725} C_VEL
LIN {X 0,Y 474.701,Z 260.982,A -85,B 0,C 180,E1 -7190.628,E2 -7190.628} C_VEL
LIN {X 0,Y 474.747,Z 260.976,A -85,B 0,C 180,E1 -7193.2,E2 -7193.2} C_VEL
LIN {X 0,Y 474.618,Z 260.991,A -85,B 0,C 180,E1 -7195.755,E2 -7195.755} C_VEL
LIN {X 0,Y 474.891,Z 260.957,A -85,B 0,C 180,E1 -7197.456,E2 -7197.456} C_VEL
LIN {X 0,Y 474.907,Z 260.954,A -85,B 0,C 180,E1 -7200.001,E2 -7200.001} C_VEL
LIN {X 0,Y 474.89,Z 260.958,A -85,B 0,C 180,E1 -7202.546,E2 -7202.546} C_VEL
LIN {X 0,Y 474.776,Z 260.97,A -85,B 0,C 180,E1 -7205.948,E2 -7205.948} C_VEL
LIN {X 0,Y 474.725,Z 260.977,A -85,B 0,C 180,E1 -7208.514,E2 -7208.514} C_VEL
LIN {X 0,Y 474.701,Z 260.982,A -85,B 0,C 180,E1 -7211.963,E2 -7211.963} C_VEL
LIN {X 0,Y 474.697,Z 260.981,A -85,B 0,C 180,E1 -7215.456,E2 -7215.456} C_VEL
LIN {X 0,Y 474.663,Z 260.985,A -85,B 0,C 180,E1 -7219.011,E2 -7219.011} C_VEL
LIN {X 0,Y 474.588,Z 260.995,A -85,B 0,C 180,E1 -7221.73,E2 -7221.73} C_VEL
LIN {X 0,Y 474.657,Z 260.988,A -85,B 0,C 180,E1 -7224.494,E2 -7224.494} C_VEL
LIN {X 0,Y 474.697,Z 260.98,A -85,B 0,C 180,E1 -7227.339,E2 -7227.339} C_VEL
LIN {X 0,Y 474.602,Z 260.996,A -85,B 0,C 180,E1 -7230.811,E2 -7230.811} C_VEL
LIN {X 0,Y 474.635,Z 260.994,A -85,B 0,C 180,E1 -7233.985,E2 -7233.985} C_VEL
LIN {X 0,Y 474.57,Z 261.001,A -85,B 0,C 180,E1 -7236.9,E2 -7236.9} C_VEL
LIN {X 0,Y 474.626,Z 260.994,A -85,B 0,C 180,E1 -7239.648,E2 -7239.648} C_VEL
LIN {X 0,Y 474.61,Z 261.066,A -85,B 0,C 180,E1 -7242.357,E2 -7242.357} C_VEL
LIN {X 0,Y 475.577,Z 266.176,A -85,B 0,C 180,E1 -7245.181,E2 -7245.181} C_VEL
LIN {X 0,Y 476.341,Z 270.845,A -85,B 0,C 180,E1 -7247.537,E2 -7247.537} C_VEL
LIN {X 0,Y 476.415,Z 275.028,A -85,B 0,C 180,E1 -7249.529,E2 -7249.529} C_VEL
LIN {X 0,Y 476.134,Z 281.289,A -85,B 0,C 180,E1 -7252.226,E2 -7252.226} C_VEL
LIN {X 0,Y 475.73,Z 288.894,A -85,B 0,C 180,E1 -7255.337,E2 -7255.337} C_VEL
LIN {X 0,Y 475.472,Z 295.318,A -85,B 0,C 180,E1 -7257.852,E2 -7257.852} C_VEL
LIN {X 0,Y 475.259,Z 303.057,A -85,B 0,C 180,E1 -7260.792,E2 -7260.792} C_VEL
LIN {X 0,Y 475.007,Z 312.381,A -85,B 0,C 180,E1 -7264.122,E2 -7264.122} C_VEL
LIN {X 0,Y 474.71,Z 321.609,A -85,B 0,C 180,E1 -7267.362,E2 -7267.362} C_VEL
LIN {X 0,Y 474.642,Z 325.076,A -85,B 0,C 180,E1 -7268.554,E2 -7268.554} C_VEL
LIN {X 0,Y 479.031,Z 342.344,A -85,B 0,C 180,E1 -7269.108,E2 -7269.108} C_VEL
LIN {X 0,Y 480.521,Z 349.617,A -85,B 0,C 180,E1 -7269.385,E2 -7269.385} C_VEL
LIN {X 0,Y 480.005,Z 363.638,A -85,B 0,C 180,E1 -7269.894,E2 -7269.894} C_VEL
LIN {X 0,Y 479.377,Z 376.821,A -85,B 0,C 180,E1 -7270.517,E2 -7270.517} C_VEL
LIN {X 0,Y 478.658,Z 389.52,A -85,B 0,C 180,E1 -7271.266,E2 -7271.266} C_VEL
LIN {X 0,Y 477.875,Z 402.804,A -85,B 0,C 180,E1 -7272.233,E2 -7272.233} C_VEL
LIN {X 0,Y 477.083,Z 414.961,A -85,B 0,C 180,E1 -7273.301,E2 -7273.301} C_VEL
LIN {X 0,Y 476.272,Z 427.188,A -85,B 0,C 180,E1 -7274.597,E2 -7274.597} C_VEL
LIN {X 0,Y 475.672,Z 437.396,A -85,B 0,C 180,E1 -7275.891,E2 -7275.891} C_VEL
LIN {X 0,Y 474.982,Z 447.489,A -85,B 0,C 180,E1 -7277.414,E2 -7277.414} C_VEL
LIN {X 0,Y 474.635,Z 455.651,A -85,B 0,C 180,E1 -7278.902,E2 -7278.902} C_VEL
LIN {X 0,Y 474.198,Z 463.426,A -85,B 0,C 180,E1 -7280.618,E2 -7280.618} C_VEL
LIN {X 0,Y 473.955,Z 469.608,A -85,B 0,C 180,E1 -7282.331,E2 -7282.331} C_VEL
LIN {X 0,Y 473.855,Z 474.387,A -85,B 0,C 180,E1 -7284.041,E2 -7284.041} C_VEL
LIN {X 0,Y 473.706,Z 477.888,A -85,B 0,C 180,E1 -7285.746,E2 -7285.746} C_VEL
LIN {X 0,Y 473.718,Z 480.19,A -85,B 0,C 180,E1 -7287.45,E2 -7287.45} C_VEL
LIN {X 0,Y 473.685,Z 481.348,A -85,B 0,C 180,E1 -7289.15,E2 -7289.15} C_VEL
LIN {X 0,Y 473.685,Z 481.347,A -85,B 0,C 180,E1 -7290.851,E2 -7290.851} C_VEL
LIN {X 0,Y 473.719,Z 480.185,A -85,B 0,C 180,E1 -7292.552,E2 -7292.552} C_VEL
LIN {X 0,Y 473.706,Z 477.882,A -85,B 0,C 180,E1 -7294.255,E2 -7294.255} C_VEL
LIN {X 0,Y 473.834,Z 474.385,A -85,B 0,C 180,E1 -7295.96,E2 -7295.96} C_VEL
LIN {X 0,Y 473.956,Z 469.607,A -85,B 0,C 180,E1 -7297.67,E2 -7297.67} C_VEL
LIN {X 0,Y 474.199,Z 463.417,A -85,B 0,C 180,E1 -7299.383,E2 -7299.383} C_VEL
LIN {X 0,Y 474.634,Z 455.639,A -85,B 0,C 180,E1 -7301.099,E2 -7301.099} C_VEL
LIN {X 0,Y 474.97,Z 447.906,A -85,B 0,C 180,E1 -7302.515,E2 -7302.515} C_VEL
LIN {X 0,Y 475.683,Z 437.387,A -85,B 0,C 180,E1 -7304.11,E2 -7304.11} C_VEL
LIN {X 0,Y 476.258,Z 427.179,A -85,B 0,C 180,E1 -7305.404,E2 -7305.404} C_VEL
LIN {X 0,Y 477.034,Z 415.547,A -85,B 0,C 180,E1 -7306.641,E2 -7306.641} C_VEL
LIN {X 0,Y 477.847,Z 402.795,A -85,B 0,C 180,E1 -7307.77,E2 -7307.77} C_VEL
LIN {X 0,Y 478.642,Z 389.495,A -85,B 0,C 180,E1 -7308.736,E2 -7308.736} C_VEL
LIN {X 0,Y 479.344,Z 376.795,A -85,B 0,C 180,E1 -7309.485,E2 -7309.485} C_VEL
LIN {X 0,Y 480.044,Z 361.86,A -85,B 0,C 180,E1 -7310.182,E2 -7310.182} C_VEL
LIN {X 0,Y 480.479,Z 348.794,A -85,B 0,C 180,E1 -7310.642,E2 -7310.642} C_VEL
LIN {X 0,Y 476.624,Z 332.884,A -85,B 0,C 180,E1 -7311.217,E2 -7311.217} C_VEL
LIN {X 0,Y 474.645,Z 325.056,A -85,B 0,C 180,E1 -7311.47,E2 -7311.47} C_VEL
LIN {X 0,Y 474.916,Z 315.25,A -85,B 0,C 180,E1 -7314.946,E2 -7314.946} C_VEL
LIN {X 0,Y 475.144,Z 307.343,A -85,B 0,C 180,E1 -7317.797,E2 -7317.797} C_VEL
LIN {X 0,Y 475.441,Z 298.741,A -85,B 0,C 180,E1 -7320.978,E2 -7320.978} C_VEL
LIN {X 0,Y 475.773,Z 290.683,A -85,B 0,C 180,E1 -7324.185,E2 -7324.185} C_VEL
LIN {X 0,Y 476.161,Z 283.238,A -85,B 0,C 180,E1 -7327.24,E2 -7327.24} C_VEL
LIN {X 0,Y 476.459,Z 276.969,A -85,B 0,C 180,E1 -7329.912,E2 -7329.912} C_VEL
LIN {X 0,Y 476.556,Z 273.268,A -85,B 0,C 180,E1 -7331.578,E2 -7331.578} C_VEL
LIN {X 0,Y 476.059,Z 268.866,A -85,B 0,C 180,E1 -7333.665,E2 -7333.665} C_VEL
LIN {X 0,Y 475.055,Z 263.389,A -85,B 0,C 180,E1 -7336.462,E2 -7336.462} C_VEL
LIN {X 0,Y 474.633,Z 260.99,A -85,B 0,C 180,E1 -7337.763,E2 -7337.763} C_VEL
LIN {X 0,Y 474.65,Z 260.988,A -85,B 0,C 180,E1 -7340.454,E2 -7340.454} C_VEL
LIN {X 0,Y 474.594,Z 260.995,A -85,B 0,C 180,E1 -7343.676,E2 -7343.676} C_VEL
LIN {X 0,Y 474.63,Z 260.992,A -85,B 0,C 180,E1 -7346.778,E2 -7346.778} C_VEL
LIN {X 0,Y 474.61,Z 260.991,A -85,B 0,C 180,E1 -7349.77,E2 -7349.77} C_VEL
LIN {X 0,Y 474.703,Z 260.981,A -85,B 0,C 180,E1 -7352.68,E2 -7352.68} C_VEL
LIN {X 0,Y 474.663,Z 260.984,A -85,B 0,C 180,E1 -7355.507,E2 -7355.507} C_VEL
LIN {X 0,Y 474.676,Z 260.984,A -85,B 0,C 180,E1 -7359.185,E2 -7359.185} C_VEL
LIN {X 0,Y 474.663,Z 260.984,A -85,B 0,C 180,E1 -7361.884,E2 -7361.884} C_VEL
LIN {X 0,Y 474.706,Z 260.982,A -85,B 0,C 180,E1 -7364.544,E2 -7364.544} C_VEL
LIN {X 0,Y 474.71,Z 260.98,A -85,B 0,C 180,E1 -7368.037,E2 -7368.037} C_VEL
LIN {X 0,Y 474.732,Z 260.975,A -85,B 0,C 180,E1 -7371.486,E2 -7371.486} C_VEL
LIN {X 0,Y 474.751,Z 260.975,A -85,B 0,C 180,E1 -7374.903,E2 -7374.903} C_VEL
LIN {X 0,Y 474.898,Z 260.954,A -85,B 0,C 180,E1 -7377.455,E2 -7377.455} C_VEL
LIN {X 0,Y 474.916,Z 260.954,A -85,B 0,C 180,E1 -7379.999,E2 -7379.999} C_VEL
LIN {X 0,Y 474.896,Z 260.957,A -85,B 0,C 180,E1 -7382.544,E2 -7382.544} C_VEL
LIN {X 0,Y 474.781,Z 260.971,A -85,B 0,C 180,E1 -7385.947,E2 -7385.947} C_VEL
LIN {X 0,Y 474.731,Z 260.979,A -85,B 0,C 180,E1 -7388.512,E2 -7388.512} C_VEL
LIN {X 0,Y 474.707,Z 260.981,A -85,B 0,C 180,E1 -7391.961,E2 -7391.961} C_VEL
LIN {X 0,Y 474.702,Z 260.979,A -85,B 0,C 180,E1 -7395.454,E2 -7395.454} C_VEL
LIN {X 0,Y 474.666,Z 260.984,A -85,B 0,C 180,E1 -7399.009,E2 -7399.009} C_VEL
LIN {X 0,Y 474.589,Z 260.995,A -85,B 0,C 180,E1 -7401.728,E2 -7401.728} C_VEL
LIN {X 0,Y 474.659,Z 260.986,A -85,B 0,C 180,E1 -7404.492,E2 -7404.492} C_VEL
LIN {X 0,Y 474.698,Z 260.98,A -85,B 0,C 180,E1 -7407.337,E2 -7407.337} C_VEL
LIN {X 0,Y 474.603,Z 260.991,A -85,B 0,C 180,E1 -7410.809,E2 -7410.809} C_VEL
LIN {X 0,Y 474.636,Z 260.99,A -85,B 0,C 180,E1 -7413.983,E2 -7413.983} C_VEL
LIN {X 0,Y 474.572,Z 260.995,A -85,B 0,C 180,E1 -7416.899,E2 -7416.899} C_VEL
LIN {X 0,Y 474.624,Z 260.991,A -85,B 0,C 180,E1 -7419.646,E2 -7419.646} C_VEL
LIN {X 0,Y 474.631,Z 260.988,A -85,B 0,C 180,E1 -7422.931,E2 -7422.931} C_VEL
LIN {X 0,Y 474.613,Z 260.993,A -85,B 0,C 180,E1 -7425.895,E2 -7425.895} C_VEL
LIN {X 0,Y 474.64,Z 260.986,A -85,B 0,C 180,E1 -7429.037,E2 -7429.037} C_VEL
LIN {X 0,Y 474.61,Z 260.993,A -85,B 0,C 180,E1 -7431.702,E2 -7431.702} C_VEL
LIN {X 0,Y 474.623,Z 260.989,A -85,B 0,C 180,E1 -7434.725,E2 -7434.725} C_VEL
LIN {X 0,Y 474.63,Z 260.991,A -85,B 0,C 180,E1 -7437.787,E2 -7437.787} C_VEL
LIN {X 0,Y 474.624,Z 260.989,A -85,B 0,C 180,E1 -7440.882,E2 -7440.882} C_VEL
LIN {X 0,Y 474.658,Z 260.987,A -85,B 0,C 180,E1 -7443.628,E2 -7443.628} C_VEL
LIN {X 0,Y 474.626,Z 260.987,A -85,B 0,C 180,E1 -7446.64,E2 -7446.64} C_VEL
LIN {X 0,Y 474.647,Z 260.987,A -85,B 0,C 180,E1 -7450.089,E2 -7450.089} C_VEL
LIN {X 0,Y 474.646,Z 260.988,A -85,B 0,C 180,E1 -7451.669,E2 -7451.669} C_VEL
LIN {X 0,Y 473.983,Z 261.07,A -85,B 0,C 180,E1 -7452.378,E2 -7452.378} C_VEL
LIN {X 0,Y 471.134,Z 261.427,A -85,B 0,C 180,E1 -7453.53,E2 -7453.53} C_VEL
LIN {X 0,Y 468.718,Z 261.728,A -85,B 0,C 180,E1 -7454.458,E2 -7454.458} C_VEL
LIN {X 0,Y 467.677,Z 261.856,A -85,B 0,C 180,E1 -7455.175,E2 -7455.175} C_VEL
LIN {X 0,Y 467.59,Z 261.866,A -85,B 0,C 180,E1 -7455.418,E2 -7455.418} C_VEL
LIN {X 0,Y 467.664,Z 261.857,A -85,B 0,C 180,E1 -7458.734,E2 -7458.734} C_VEL
LIN {X 0,Y 467.738,Z 261.846,A -85,B 0,C 180,E1 -7462.228,E2 -7462.228} C_VEL
LIN {X 0,Y 467.693,Z 261.853,A -85,B 0,C 180,E1 -7464.827,E2 -7464.827} C_VEL
LIN {X 0,Y 467.369,Z 261.897,A -85,B 0,C 180,E1 -7468.276,E2 -7468.276} C_VEL
LIN {X 0,Y 467.568,Z 262.511,A -85,B 0,C 180,E1 -7469.138,E2 -7469.138} C_VEL
LIN {X 0,Y 467.33,Z 264.111,A -85,B 0,C 180,E1 -7470.861,E2 -7470.861} C_VEL
LIN {X 0,Y 467.197,Z 267.284,A -85,B 0,C 180,E1 -7474.313,E2 -7474.313} C_VEL
LIN {X 0,Y 467.1,Z 269.708,A -85,B 0,C 180,E1 -7476.913,E2 -7476.913} C_VEL
LIN {X 0,Y 466.939,Z 273.015,A -85,B 0,C 180,E1 -7480.405,E2 -7480.405} C_VEL
LIN {X 0,Y 467.014,Z 273.865,A -85,B 0,C 180,E1 -7481.324,E2 -7481.324} C_VEL
LIN {X 0,Y 471.964,Z 289.511,A -85,B 0,C 180,E1 -7481.932,E2 -7481.932} C_VEL
LIN {X 0,Y 473.881,Z 296.606,A -85,B 0,C 180,E1 -7482.252,E2 -7482.252} C_VEL
LIN {X 0,Y 473.336,Z 310.233,A -85,B 0,C 180,E1 -7482.783,E2 -7482.783} C_VEL
LIN {X 0,Y 472.658,Z 324.071,A -85,B 0,C 180,E1 -7483.488,E2 -7483.488} C_VEL
LIN {X 0,Y 471.95,Z 337.37,A -85,B 0,C 180,E1 -7484.341,E2 -7484.341} C_VEL
LIN {X 0,Y 471.182,Z 350.253,A -85,B 0,C 180,E1 -7485.352,E2 -7485.352} C_VEL
LIN {X 0,Y 470.39,Z 362.286,A -85,B 0,C 180,E1 -7486.491,E2 -7486.491} C_VEL
LIN {X 0,Y 469.611,Z 372.549,A -85,B 0,C 180,E1 -7487.64,E2 -7487.64} C_VEL
LIN {X 0,Y 469.029,Z 381.381,A -85,B 0,C 180,E1 -7488.793,E2 -7488.793} C_VEL
LIN {X 0,Y 468.303,Z 391.813,A -85,B 0,C 180,E1 -7490.421,E2 -7490.421} C_VEL
LIN {X 0,Y 467.751,Z 400.454,A -85,B 0,C 180,E1 -7492.062,E2 -7492.062} C_VEL
LIN {X 0,Y 467.425,Z 406.66,A -85,B 0,C 180,E1 -7493.488,E2 -7493.488} C_VEL
LIN {X 0,Y 467.132,Z 411.82,A -85,B 0,C 180,E1 -7494.913,E2 -7494.913} C_VEL
LIN {X 0,Y 466.959,Z 416.127,A -85,B 0,C 180,E1 -7496.358,E2 -7496.358} C_VEL
LIN {X 0,Y 466.77,Z 419.495,A -85,B 0,C 180,E1 -7497.823,E2 -7497.823} C_VEL
LIN {X 0,Y 466.672,Z 421.842,A -85,B 0,C 180,E1 -7499.139,E2 -7499.139} C_VEL
LIN {X 0,Y 466.613,Z 423.813,A -85,B 0,C 180,E1 -7500.852,E2 -7500.852} C_VEL
LIN {X 0,Y 466.567,Z 424.741,A -85,B 0,C 180,E1 -7502.838,E2 -7502.838} C_VEL
LIN {X 0,Y 466.593,Z 424.589,A -85,B 0,C 180,E1 -7504.065,E2 -7504.065} C_VEL
LIN {X 0,Y 466.615,Z 423.203,A -85,B 0,C 180,E1 -7505.972,E2 -7505.972} C_VEL
LIN {X 0,Y 466.648,Z 421.8,A -85,B 0,C 180,E1 -7507.043,E2 -7507.043} C_VEL
LIN {X 0,Y 466.849,Z 419.192,A -85,B 0,C 180,E1 -7508.483,E2 -7508.483} C_VEL
LIN {X 0,Y 467.032,Z 414.656,A -85,B 0,C 180,E1 -7510.32,E2 -7510.32} C_VEL
LIN {X 0,Y 467.299,Z 409.219,A -85,B 0,C 180,E1 -7511.994,E2 -7511.994} C_VEL
LIN {X 0,Y 467.662,Z 402.123,A -85,B 0,C 180,E1 -7513.731,E2 -7513.731} C_VEL
LIN {X 0,Y 468.228,Z 394.218,A -85,B 0,C 180,E1 -7515.302,E2 -7515.302} C_VEL
LIN {X 0,Y 468.819,Z 385.332,A -85,B 0,C 180,E1 -7516.774,E2 -7516.774} C_VEL
LIN {X 0,Y 469.548,Z 374.951,A -85,B 0,C 180,E1 -7518.209,E2 -7518.209} C_VEL
LIN {X 0,Y 470.38,Z 363.553,A -85,B 0,C 180,E1 -7519.521,E2 -7519.521} C_VEL
